   DATA[1018,16] := 1.0;
   DATA[1018,17] := 1.0;
   DATA[1018,18] := 1.0;
   DATA[1018,19] := 1.0;
   DATA[1018,20] := 148.808;
   DATA[1018,21] := 155.0115;
   DATA[1018,22] := 1.715567;
   DATA[1018,23] := 905.2679;
   DATA[1018,24] := 2.0;
   DATA[1018,25] := 2.0;
   DATA[1018,26] := 7.87798;
   DATA[1018,27] := 144.1169;
   DATA[1018,28] := 263.1056;
   DATA[1018,29] := 12.03538;
   DATA[1018,30] := 1.72443;
   DATA[1018,31] := 1.268093;
   DATA[1018,32] := 0.7351407;
   DATA[1018,33] := 0.3083624;
   DATA[1018,34] := 2.0;
   DATA[1018,35] := 250.1442;
   DATA[1018,36] := 1.649953;
   DATA[1018,37] := 189.1022;
   DATA[1018,38] := 0.000128152;
   DATA[1018,39] := 1.0;
   DATA[1019,0] := 2.541075;
   DATA[1019,1] := 664.7062;
   DATA[1019,2] := 2.0;
   DATA[1019,3] := 1.0;
   DATA[1019,4] := 262.5288;
   DATA[1019,5] := 8.462126;
   DATA[1019,6] := 315.9959;
   DATA[1019,8] := 1.0;
   DATA[1019,9] := 1.0;
   DATA[1019,10] := 1.0;
   DATA[1019,11] := 2.010372;
   DATA[1019,13] := 1011.439;
   DATA[1019,14] := 1.0;
   DATA[1019,15] := 1.0;
   DATA[1019,16] := 1.0;
   DATA[1019,17] := 1.0;
   DATA[1019,18] := 1.0;
   DATA[1019,19] := 1.0;
   DATA[1019,20] := 148.808;
   DATA[1019,21] := 155.0115;
   DATA[1019,22] := 1.715567;
   DATA[1019,23] := 904.8449;
   DATA[1019,24] := 2.0;
   DATA[1019,25] := 2.0;
   DATA[1019,26] := 7.87798;
   DATA[1019,27] := 144.0913;
   DATA[1019,28] := 263.1056;
   DATA[1019,29] := 12.03538;
   DATA[1019,30] := 1.72443;
   DATA[1019,31] := 1.265531;
   DATA[1019,32] := 0.7351407;
   DATA[1019,33] := 0.3083624;
   DATA[1019,34] := 2.0;
   DATA[1019,35] := 250.1442;
   DATA[1019,36] := 1.649953;
   DATA[1019,37] := 189.0541;
   DATA[1019,38] := 0.000128152;
   DATA[1019,39] := 1.0;
   DATA[1020,0] := 2.541075;
   DATA[1020,1] := 665.4913;
   DATA[1020,2] := 2.0;
   DATA[1020,3] := 1.0;
   DATA[1020,4] := 262.5288;
   DATA[1020,5] := 8.462126;
   DATA[1020,6] := 315.9959;
   DATA[1020,8] := 1.0;
   DATA[1020,9] := 1.0;
   DATA[1020,10] := 1.0;
   DATA[1020,11] := 2.010372;
   DATA[1020,13] := 1011.279;
   DATA[1020,14] := 1.0;
   DATA[1020,15] := 1.0;
   DATA[1020,16] := 1.0;
   DATA[1020,17] := 1.0;
   DATA[1020,18] := 1.0;
   DATA[1020,19] := 1.0;
   DATA[1020,20] := 148.808;
   DATA[1020,21] := 155.0115;
   DATA[1020,22] := 1.713645;
   DATA[1020,23] := 904.3835;
   DATA[1020,24] := 2.0;
   DATA[1020,25] := 2.0;
   DATA[1020,26] := 7.87798;
   DATA[1020,27] := 144.0913;
   DATA[1020,28] := 263.1056;
   DATA[1020,29] := 12.03538;
   DATA[1020,30] := 1.72443;
   DATA[1020,31] := 1.28436;
   DATA[1020,32] := 0.7351407;
   DATA[1020,33] := 0.3083624;
   DATA[1020,34] := 2.0;
   DATA[1020,35] := 250.1442;
   DATA[1020,36] := 1.665972;
   DATA[1020,37] := 189.0541;
   DATA[1020,38] := 0.000128152;
   DATA[1020,39] := 1.0;
   DATA[1021,0] := 2.542356;
   DATA[1021,1] := 666.4333;
   DATA[1021,2] := 2.0;
   DATA[1021,3] := 1.0;
   DATA[1021,4] := 262.5288;
   DATA[1021,5] := 8.462126;
   DATA[1021,6] := 315.8165;
   DATA[1021,8] := 1.0;
   DATA[1021,9] := 1.0;
   DATA[1021,10] := 1.0;
   DATA[1021,11] := 2.010372;
   DATA[1021,13] := 1011.279;
   DATA[1021,14] := 1.0;
   DATA[1021,15] := 1.0;
   DATA[1021,16] := 1.0;
   DATA[1021,17] := 1.0;
   DATA[1021,18] := 1.0;
   DATA[1021,19] := 1.0;
   DATA[1021,20] := 148.808;
   DATA[1021,21] := 155.0115;
   DATA[1021,22] := 1.713645;
   DATA[1021,23] := 903.8452;
   DATA[1021,24] := 2.0;
   DATA[1021,25] := 2.0;
   DATA[1021,26] := 7.87798;
   DATA[1021,27] := 144.0913;
   DATA[1021,28] := 263.1056;
   DATA[1021,29] := 12.03538;
   DATA[1021,30] := 1.72443;
   DATA[1021,31] := 1.292174;
   DATA[1021,32] := 0.7351407;
   DATA[1021,33] := 0.3083624;
   DATA[1021,34] := 2.0;
   DATA[1021,35] := 250.4005;
   DATA[1021,36] := 1.665972;
   DATA[1021,37] := 189.0541;
   DATA[1021,38] := 0.000128152;
   DATA[1021,39] := 1.0;
   DATA[1022,0] := 2.54588;
   DATA[1022,1] := 666.5511;
   DATA[1022,2] := 2.0;
   DATA[1022,3] := 1.0;
   DATA[1022,4] := 262.5288;
   DATA[1022,5] := 8.462126;
   DATA[1022,6] := 315.8165;
   DATA[1022,8] := 1.0;
   DATA[1022,9] := 1.0;
   DATA[1022,10] := 1.0;
   DATA[1022,11] := 2.010372;
   DATA[1022,13] := 1011.119;
   DATA[1022,14] := 1.0;
   DATA[1022,15] := 1.0;
   DATA[1022,16] := 1.0;
   DATA[1022,17] := 1.0;
   DATA[1022,18] := 1.0;
   DATA[1022,19] := 1.0;
   DATA[1022,20] := 148.808;
   DATA[1022,21] := 155.0115;
   DATA[1022,22] := 1.713645;
   DATA[1022,23] := 903.6913;
   DATA[1022,24] := 2.0;
   DATA[1022,25] := 2.0;
   DATA[1022,26] := 7.87798;
   DATA[1022,27] := 144.0913;
   DATA[1022,28] := 263.1056;
   DATA[1022,29] := 12.03538;
   DATA[1022,30] := 1.72443;
   DATA[1022,31] := 1.292174;
   DATA[1022,32] := 0.7351407;
   DATA[1022,33] := 0.3083624;
   DATA[1022,34] := 2.0;
   DATA[1022,35] := 250.4005;
   DATA[1022,36] := 1.69801;
   DATA[1022,37] := 189.1823;
   DATA[1022,38] := 0.000128152;
   DATA[1022,39] := 1.0;
   DATA[1023,0] := 2.54588;
   DATA[1023,1] := 667.3361;
   DATA[1023,2] := 2.0;
   DATA[1023,3] := 1.0;
   DATA[1023,4] := 262.5288;
   DATA[1023,5] := 8.462126;
   DATA[1023,6] := 315.8165;
   DATA[1023,8] := 1.0;
   DATA[1023,9] := 1.0;
   DATA[1023,10] := 1.0;
   DATA[1023,11] := 2.010372;
   DATA[1023,13] := 1011.239;
   DATA[1023,14] := 1.0;
   DATA[1023,15] := 1.0;
   DATA[1023,16] := 1.0;
   DATA[1023,17] := 1.0;
   DATA[1023,18] := 1.0;
   DATA[1023,19] := 1.0;
   DATA[1023,20] := 148.808;
   DATA[1023,21] := 155.0115;
   DATA[1023,22] := 1.716592;
   DATA[1023,23] := 903.2299;
   DATA[1023,24] := 2.0;
   DATA[1023,25] := 2.0;
   DATA[1023,26] := 7.87798;
   DATA[1023,27] := 144.0913;
   DATA[1023,28] := 263.1056;
   DATA[1023,29] := 12.03538;
   DATA[1023,30] := 1.728531;
   DATA[1023,31] := 1.292174;
   DATA[1023,32] := 0.7351407;
   DATA[1023,33] := 0.3083624;
   DATA[1023,34] := 2.0;
   DATA[1023,35] := 250.5608;
   DATA[1023,36] := 1.730048;
   DATA[1023,37] := 189.3425;
   DATA[1023,38] := 0.000128152;
   DATA[1023,39] := 1.0;
   DATA[1024,0] := 2.54588;
   DATA[1024,1] := 667.6894;
   DATA[1024,2] := 2.0;
   DATA[1024,3] := 1.0;
   DATA[1024,4] := 262.5288;
   DATA[1024,5] := 8.462126;
   DATA[1024,6] := 315.9446;
   DATA[1024,8] := 1.0;
   DATA[1024,9] := 1.0;
   DATA[1024,10] := 1.0;
   DATA[1024,11] := 2.010372;
   DATA[1024,13] := 1011.56;
   DATA[1024,14] := 1.0;
   DATA[1024,15] := 1.0;
   DATA[1024,16] := 1.0;
   DATA[1024,17] := 1.0;
   DATA[1024,18] := 1.0;
   DATA[1024,19] := 1.0;
   DATA[1024,20] := 148.808;
   DATA[1024,21] := 154.8065;
   DATA[1024,22] := 1.717746;
   DATA[1024,23] := 903.0761;
   DATA[1024,24] := 2.0;
   DATA[1024,25] := 2.0;
   DATA[1024,26] := 7.87798;
   DATA[1024,27] := 144.0913;
   DATA[1024,28] := 263.1056;
   DATA[1024,29] := 12.03538;
   DATA[1024,30] := 1.728531;
   DATA[1024,31] := 1.292174;
   DATA[1024,32] := 0.7351407;
   DATA[1024,33] := 0.3071454;
   DATA[1024,34] := 2.0;
   DATA[1024,35] := 250.5608;
   DATA[1024,36] := 1.730048;
   DATA[1024,37] := 189.3425;
   DATA[1024,38] := 0.000128152;
   DATA[1024,39] := 1.0;
   DATA[1025,0] := 2.54588;
   DATA[1025,1] := 667.6501;
   DATA[1025,2] := 2.0;
   DATA[1025,3] := 1.0;
   DATA[1025,4] := 262.5288;
   DATA[1025,5] := 8.462126;
   DATA[1025,6] := 315.9446;
   DATA[1025,8] := 1.0;
   DATA[1025,9] := 1.0;
   DATA[1025,10] := 1.0;
   DATA[1025,11] := 2.010372;
   DATA[1025,13] := 1011.56;
   DATA[1025,14] := 1.0;
   DATA[1025,15] := 1.0;
   DATA[1025,16] := 1.0;
   DATA[1025,17] := 1.0;
   DATA[1025,18] := 1.0;
   DATA[1025,19] := 1.0;
   DATA[1025,20] := 148.808;
   DATA[1025,21] := 154.8065;
   DATA[1025,22] := 1.717746;
   DATA[1025,23] := 902.4609;
   DATA[1025,24] := 2.0;
   DATA[1025,25] := 2.0;
   DATA[1025,26] := 7.87798;
   DATA[1025,27] := 144.0913;
   DATA[1025,28] := 263.1056;
   DATA[1025,29] := 12.03538;
   DATA[1025,30] := 1.726865;
   DATA[1025,31] := 1.292174;
   DATA[1025,32] := 0.7351407;
   DATA[1025,33] := 0.3068891;
   DATA[1025,34] := 2.0;
   DATA[1025,35] := 250.5608;
   DATA[1025,36] := 1.730048;
   DATA[1025,37] := 189.3425;
   DATA[1025,38] := 0.000128152;
   DATA[1025,39] := 1.0;
   DATA[1026,0] := 2.54588;
   DATA[1026,1] := 668.1997;
   DATA[1026,2] := 2.0;
   DATA[1026,3] := 1.0;
   DATA[1026,4] := 262.5288;
   DATA[1026,5] := 8.46501;
   DATA[1026,6] := 315.9446;
   DATA[1026,8] := 1.0;
   DATA[1026,9] := 1.0;
   DATA[1026,10] := 1.0;
   DATA[1026,11] := 2.010372;
   DATA[1026,13] := 1011.159;
   DATA[1026,14] := 1.0;
   DATA[1026,15] := 1.0;
   DATA[1026,16] := 1.0;
   DATA[1026,17] := 1.0;
   DATA[1026,18] := 1.0;
   DATA[1026,19] := 1.0;
   DATA[1026,20] := 148.808;
   DATA[1026,21] := 154.8065;
   DATA[1026,22] := 1.717746;
   DATA[1026,23] := 901.7688;
   DATA[1026,24] := 2.0;
   DATA[1026,25] := 2.0;
   DATA[1026,26] := 7.87798;
   DATA[1026,27] := 144.0913;
   DATA[1026,28] := 263.1056;
   DATA[1026,29] := 12.03538;
   DATA[1026,30] := 1.726224;
   DATA[1026,31] := 1.300243;
   DATA[1026,32] := 0.7351407;
   DATA[1026,33] := 0.3068891;
   DATA[1026,34] := 2.0;
   DATA[1026,35] := 250.721;
   DATA[1026,36] := 1.730048;
   DATA[1026,37] := 189.3425;
   DATA[1026,38] := 0.000128152;
   DATA[1026,39] := 1.0;
   DATA[1027,0] := 2.539474;
   DATA[1027,1] := 668.3174;
   DATA[1027,2] := 2.0;
   DATA[1027,3] := 1.0;
   DATA[1027,4] := 262.5288;
   DATA[1027,5] := 8.46501;
   DATA[1027,6] := 315.9446;
   DATA[1027,8] := 1.0;
   DATA[1027,9] := 1.0;
   DATA[1027,10] := 1.0;
   DATA[1027,11] := 2.010372;
   DATA[1027,13] := 1010.959;
   DATA[1027,14] := 1.0;
   DATA[1027,15] := 1.0;
   DATA[1027,16] := 1.0;
   DATA[1027,17] := 1.0;
   DATA[1027,18] := 1.0;
   DATA[1027,19] := 1.0;
   DATA[1027,20] := 148.808;
   DATA[1027,21] := 154.8065;
   DATA[1027,22] := 1.718643;
   DATA[1027,23] := 901.1536;
   DATA[1027,24] := 2.0;
   DATA[1027,25] := 2.0;
   DATA[1027,26] := 7.87798;
   DATA[1027,27] := 144.0913;
   DATA[1027,28] := 263.1056;
   DATA[1027,29] := 12.03538;
   DATA[1027,30] := 1.726224;
   DATA[1027,31] := 1.296657;
   DATA[1027,32] := 0.7351407;
   DATA[1027,33] := 0.3068891;
   DATA[1027,34] := 2.0;
   DATA[1027,35] := 250.753;
   DATA[1027,36] := 1.730048;
   DATA[1027,37] := 189.3425;
   DATA[1027,38] := 0.000128152;
   DATA[1027,39] := 1.0;
   DATA[1028,0] := 2.536912;
   DATA[1028,1] := 668.239;
   DATA[1028,2] := 2.0;
   DATA[1028,3] := 1.0;
   DATA[1028,4] := 262.5288;
   DATA[1028,5] := 8.46501;
   DATA[1028,6] := 315.9446;
   DATA[1028,8] := 1.0;
   DATA[1028,9] := 1.0;
   DATA[1028,10] := 1.0;
   DATA[1028,11] := 2.010372;
   DATA[1028,13] := 1011.039;
   DATA[1028,14] := 1.0;
   DATA[1028,15] := 1.0;
   DATA[1028,16] := 1.0;
   DATA[1028,17] := 1.0;
   DATA[1028,18] := 1.0;
   DATA[1028,19] := 1.0;
   DATA[1028,20] := 148.808;
   DATA[1028,21] := 154.8065;
   DATA[1028,22] := 1.720437;
   DATA[1028,23] := 901.0382;
   DATA[1028,24] := 2.0;
   DATA[1028,25] := 2.0;
   DATA[1028,26] := 7.87798;
   DATA[1028,27] := 144.0913;
   DATA[1028,28] := 263.1056;
   DATA[1028,29] := 12.03538;
   DATA[1028,30] := 1.726224;
   DATA[1028,31] := 1.291918;
   DATA[1028,32] := 0.7351407;
   DATA[1028,33] := 0.3068891;
   DATA[1028,34] := 2.0;
   DATA[1028,35] := 250.8011;
   DATA[1028,36] := 1.730048;
   DATA[1028,37] := 189.4867;
   DATA[1028,38] := 0.000128152;
   DATA[1028,39] := 1.0;
   DATA[1029,0] := 2.532428;
   DATA[1029,1] := 668.5137;
   DATA[1029,2] := 2.0;
   DATA[1029,3] := 1.0;
   DATA[1029,4] := 262.5288;
   DATA[1029,5] := 8.46501;
   DATA[1029,6] := 315.9446;
   DATA[1029,8] := 1.0;
   DATA[1029,9] := 1.0;
   DATA[1029,10] := 1.0;
   DATA[1029,11] := 2.010372;
   DATA[1029,13] := 1010.879;
   DATA[1029,14] := 1.0;
   DATA[1029,15] := 1.0;
   DATA[1029,16] := 1.0;
   DATA[1029,17] := 1.0;
   DATA[1029,18] := 1.0;
   DATA[1029,19] := 1.0;
   DATA[1029,20] := 148.808;
   DATA[1029,21] := 154.8065;
   DATA[1029,22] := 1.720565;
   DATA[1029,23] := 900.0769;
   DATA[1029,24] := 2.0;
   DATA[1029,25] := 2.0;
   DATA[1029,26] := 7.87798;
   DATA[1029,27] := 144.0913;
   DATA[1029,28] := 263.1056;
   DATA[1029,29] := 12.03538;
   DATA[1029,30] := 1.727634;
   DATA[1029,31] := 1.282311;
   DATA[1029,32] := 0.7351407;
   DATA[1029,33] := 0.3065689;
   DATA[1029,34] := 2.0;
   DATA[1029,35] := 250.8011;
   DATA[1029,36] := 1.730048;
   DATA[1029,37] := 189.5187;
   DATA[1029,38] := 0.000128152;
   DATA[1029,39] := 1.0;
   DATA[1030,0] := 2.532428;
   DATA[1030,1] := 669.2203;
   DATA[1030,2] := 2.0;
   DATA[1030,3] := 1.0;
   DATA[1030,4] := 262.5288;
   DATA[1030,5] := 8.46501;
   DATA[1030,6] := 315.9446;
   DATA[1030,8] := 1.0;
   DATA[1030,9] := 1.0;
   DATA[1030,10] := 1.0;
   DATA[1030,11] := 2.010372;
   DATA[1030,13] := 1010.879;
   DATA[1030,14] := 1.0;
   DATA[1030,15] := 1.0;
   DATA[1030,16] := 1.0;
   DATA[1030,17] := 1.0;
   DATA[1030,18] := 1.0;
   DATA[1030,19] := 1.0;
   DATA[1030,20] := 148.808;
   DATA[1030,21] := 154.6526;
   DATA[1030,22] := 1.720565;
   DATA[1030,23] := 899.5001;
   DATA[1030,24] := 2.0;
   DATA[1030,25] := 2.0;
   DATA[1030,26] := 7.87798;
   DATA[1030,27] := 144.0913;
   DATA[1030,28] := 263.1056;
   DATA[1030,29] := 12.03538;
   DATA[1030,30] := 1.727634;
   DATA[1030,31] := 1.281927;
   DATA[1030,32] := 0.7351407;
   DATA[1030,33] := 0.3065689;
   DATA[1030,34] := 2.0;
   DATA[1030,35] := 250.8011;
   DATA[1030,36] := 1.730048;
   DATA[1030,37] := 189.6148;
   DATA[1030,38] := 0.000128152;
   DATA[1030,39] := 1.0;
   DATA[1031,0] := 2.532428;
   DATA[1031,1] := 669.5735;
   DATA[1031,2] := 2.0;
   DATA[1031,3] := 1.0;
   DATA[1031,4] := 262.5288;
   DATA[1031,5] := 8.464048;
   DATA[1031,6] := 315.9446;
   DATA[1031,8] := 1.0;
   DATA[1031,9] := 1.0;
   DATA[1031,10] := 1.0;
   DATA[1031,11] := 2.010372;
   DATA[1031,13] := 1010.959;
   DATA[1031,14] := 1.0;
   DATA[1031,15] := 1.0;
   DATA[1031,16] := 1.0;
   DATA[1031,17] := 1.0;
   DATA[1031,18] := 1.0;
   DATA[1031,19] := 1.0;
   DATA[1031,20] := 148.808;
   DATA[1031,21] := 154.6526;
   DATA[1031,22] := 1.720565;
   DATA[1031,23] := 899.2694;
   DATA[1031,24] := 2.0;
   DATA[1031,25] := 2.0;
   DATA[1031,26] := 7.87798;
   DATA[1031,27] := 144.0913;
   DATA[1031,28] := 263.1056;
   DATA[1031,29] := 12.03538;
   DATA[1031,30] := 1.727634;
   DATA[1031,31] := 1.286922;
   DATA[1031,32] := 0.7351407;
   DATA[1031,33] := 0.3065689;
   DATA[1031,34] := 2.0;
   DATA[1031,35] := 250.8011;
   DATA[1031,36] := 1.730048;
   DATA[1031,37] := 189.6148;
   DATA[1031,38] := 0.000128152;
   DATA[1031,39] := 1.0;
   DATA[1032,0] := 2.538513;
   DATA[1032,1] := 669.652;
   DATA[1032,2] := 2.0;
   DATA[1032,3] := 1.0;
   DATA[1032,4] := 262.5288;
   DATA[1032,5] := 8.462446;
   DATA[1032,6] := 316.0728;
   DATA[1032,8] := 1.0;
   DATA[1032,9] := 1.0;
   DATA[1032,10] := 1.0;
   DATA[1032,11] := 2.010372;
   DATA[1032,13] := 1011.079;
   DATA[1032,14] := 1.0;
   DATA[1032,15] := 1.0;
   DATA[1032,16] := 1.0;
   DATA[1032,17] := 1.0;
   DATA[1032,18] := 1.0;
   DATA[1032,19] := 1.0;
   DATA[1032,20] := 148.808;
   DATA[1032,21] := 154.6526;
   DATA[1032,22] := 1.719668;
   DATA[1032,23] := 899.0002;
   DATA[1032,24] := 2.0;
   DATA[1032,25] := 2.0;
   DATA[1032,26] := 7.87798;
   DATA[1032,27] := 144.0913;
   DATA[1032,28] := 263.1056;
   DATA[1032,29] := 12.03538;
   DATA[1032,30] := 1.727634;
   DATA[1032,31] := 1.29243;
   DATA[1032,32] := 0.7351407;
   DATA[1032,33] := 0.3065689;
   DATA[1032,34] := 2.0;
   DATA[1032,35] := 250.8652;
   DATA[1032,36] := 1.730048;
   DATA[1032,37] := 189.6148;
   DATA[1032,38] := 0.000128152;
   DATA[1032,39] := 1.0;
   DATA[1033,0] := 2.543638;
   DATA[1033,1] := 670.0839;
   DATA[1033,2] := 2.0;
   DATA[1033,3] := 1.0;
   DATA[1033,4] := 262.5288;
   DATA[1033,5] := 8.461164;
   DATA[1033,6] := 316.0728;
   DATA[1033,8] := 1.0;
   DATA[1033,9] := 1.0;
   DATA[1033,10] := 1.0;
   DATA[1033,11] := 2.010372;
   DATA[1033,13] := 1010.959;
   DATA[1033,14] := 1.0;
   DATA[1033,15] := 1.0;
   DATA[1033,16] := 1.0;
   DATA[1033,17] := 1.0;
   DATA[1033,18] := 1.0;
   DATA[1033,19] := 1.0;
   DATA[1033,20] := 148.808;
   DATA[1033,21] := 154.6526;
   DATA[1033,22] := 1.718643;
   DATA[1033,23] := 898.4619;
   DATA[1033,24] := 2.0;
   DATA[1033,25] := 2.0;
   DATA[1033,26] := 7.87798;
   DATA[1033,27] := 144.0913;
   DATA[1033,28] := 263.1056;
   DATA[1033,29] := 12.03538;
   DATA[1033,30] := 1.72789;
   DATA[1033,31] := 1.29243;
   DATA[1033,32] := 0.7351407;
   DATA[1033,33] := 0.3065689;
   DATA[1033,34] := 2.0;
   DATA[1033,35] := 250.9453;
   DATA[1033,36] := 1.730048;
   DATA[1033,37] := 189.6148;
   DATA[1033,38] := 0.000128152;
   DATA[1033,39] := 1.0;
   DATA[1034,0] := 2.54684;
   DATA[1034,1] := 671.1437;
   DATA[1034,2] := 2.0;
   DATA[1034,3] := 1.0;
   DATA[1034,4] := 262.5288;
   DATA[1034,5] := 8.461164;
   DATA[1034,6] := 316.0728;
   DATA[1034,8] := 1.0;
   DATA[1034,9] := 1.0;
   DATA[1034,10] := 1.0;
   DATA[1034,11] := 2.010372;
   DATA[1034,13] := 1011.039;
   DATA[1034,14] := 1.0;
   DATA[1034,15] := 1.0;
   DATA[1034,16] := 1.0;
   DATA[1034,17] := 1.0;
   DATA[1034,18] := 1.0;
   DATA[1034,19] := 1.0;
   DATA[1034,20] := 148.808;
   DATA[1034,21] := 154.8321;
   DATA[1034,22] := 1.718643;
   DATA[1034,23] := 898.0389;
   DATA[1034,24] := 2.0;
   DATA[1034,25] := 2.0;
   DATA[1034,26] := 7.87798;
   DATA[1034,27] := 144.0913;
   DATA[1034,28] := 263.1056;
   DATA[1034,29] := 12.03538;
   DATA[1034,30] := 1.728788;
   DATA[1034,31] := 1.283592;
   DATA[1034,32] := 0.7351407;
   DATA[1034,33] := 0.3065689;
   DATA[1034,34] := 2.0;
   DATA[1034,35] := 250.9453;
   DATA[1034,36] := 1.730048;
   DATA[1034,37] := 189.6148;
   DATA[1034,38] := 0.000128152;
   DATA[1034,39] := 1.0;
   DATA[1035,0] := 2.54684;
   DATA[1035,1] := 671.811;
   DATA[1035,2] := 2.0;
   DATA[1035,3] := 1.0;
   DATA[1035,4] := 262.5288;
   DATA[1035,5] := 8.461164;
   DATA[1035,6] := 316.0728;
   DATA[1035,8] := 1.0;
   DATA[1035,9] := 1.0;
   DATA[1035,10] := 1.0;
   DATA[1035,11] := 2.010372;
   DATA[1035,13] := 1010.919;
   DATA[1035,14] := 1.0;
   DATA[1035,15] := 1.0;
   DATA[1035,16] := 1.0;
   DATA[1035,17] := 1.0;
   DATA[1035,18] := 1.0;
   DATA[1035,19] := 1.0;
   DATA[1035,20] := 148.808;
   DATA[1035,21] := 154.8321;
   DATA[1035,22] := 1.719796;
   DATA[1035,23] := 897.8467;
   DATA[1035,24] := 2.0;
   DATA[1035,25] := 2.0;
   DATA[1035,26] := 7.87798;
   DATA[1035,27] := 144.0913;
   DATA[1035,28] := 263.1056;
   DATA[1035,29] := 12.03538;
   DATA[1035,30] := 1.729428;
   DATA[1035,31] := 1.264506;
   DATA[1035,32] := 0.7351407;
   DATA[1035,33] := 0.3065689;
   DATA[1035,34] := 2.0;
   DATA[1035,35] := 250.9453;
   DATA[1035,36] := 1.730048;
   DATA[1035,37] := 189.6148;
   DATA[1035,38] := 0.000128152;
   DATA[1035,39] := 1.0;
   DATA[1036,0] := 2.550684;
   DATA[1036,1] := 672.125;
   DATA[1036,2] := 2.0;
   DATA[1036,3] := 1.0;
   DATA[1036,4] := 262.5288;
   DATA[1036,5] := 8.461164;
   DATA[1036,6] := 316.0728;
   DATA[1036,8] := 1.0;
   DATA[1036,9] := 1.0;
   DATA[1036,10] := 1.0;
   DATA[1036,11] := 2.010372;
   DATA[1036,13] := 1010.718;
   DATA[1036,14] := 1.0;
   DATA[1036,15] := 1.0;
   DATA[1036,16] := 1.0;
   DATA[1036,17] := 1.0;
   DATA[1036,18] := 1.0;
   DATA[1036,19] := 1.0;
   DATA[1036,20] := 148.808;
   DATA[1036,21] := 154.8321;
   DATA[1036,22] := 1.719796;
   DATA[1036,23] := 897.616;
   DATA[1036,24] := 2.0;
   DATA[1036,25] := 2.0;
   DATA[1036,26] := 7.87798;
   DATA[1036,27] := 144.0913;
   DATA[1036,28] := 263.1056;
   DATA[1036,29] := 12.03538;
   DATA[1036,30] := 1.729428;
   DATA[1036,31] := 1.262457;
   DATA[1036,32] := 0.7351407;
   DATA[1036,33] := 0.3065689;
   DATA[1036,34] := 2.0;
   DATA[1036,35] := 250.9453;
   DATA[1036,36] := 1.730048;
   DATA[1036,37] := 189.6148;
   DATA[1036,38] := 0.000128152;
   DATA[1036,39] := 1.0;
   DATA[1037,0] := 2.550684;
   DATA[1037,1] := 673.0278;
   DATA[1037,2] := 2.0;
   DATA[1037,3] := 1.0;
   DATA[1037,4] := 262.5288;
   DATA[1037,5] := 8.461164;
   DATA[1037,6] := 316.201;
   DATA[1037,8] := 1.0;
   DATA[1037,9] := 1.0;
   DATA[1037,10] := 1.0;
   DATA[1037,11] := 2.010372;
   DATA[1037,13] := 1011.279;
   DATA[1037,14] := 1.0;
   DATA[1037,15] := 1.0;
   DATA[1037,16] := 1.0;
   DATA[1037,17] := 1.0;
   DATA[1037,18] := 1.0;
   DATA[1037,19] := 1.0;
   DATA[1037,20] := 148.808;
   DATA[1037,21] := 154.8321;
   DATA[1037,22] := 1.719796;
   DATA[1037,23] := 897.27;
   DATA[1037,24] := 2.0;
   DATA[1037,25] := 2.0;
   DATA[1037,26] := 7.87798;
   DATA[1037,27] := 144.0913;
   DATA[1037,28] := 263.1056;
   DATA[1037,29] := 12.03538;
   DATA[1037,30] := 1.729428;
   DATA[1037,31] := 1.265147;
   DATA[1037,32] := 0.7351407;
   DATA[1037,33] := 0.3080421;
   DATA[1037,34] := 2.0;
   DATA[1037,35] := 250.753;
   DATA[1037,36] := 1.730048;
   DATA[1037,37] := 189.6148;
   DATA[1037,38] := 0.000128152;
   DATA[1037,39] := 1.0;
   DATA[1038,0] := 2.550684;
   DATA[1038,1] := 673.7343;
   DATA[1038,2] := 2.0;
   DATA[1038,3] := 1.0;
   DATA[1038,4] := 262.5288;
   DATA[1038,5] := 8.463408;
   DATA[1038,6] := 316.201;
   DATA[1038,8] := 1.0;
   DATA[1038,9] := 1.0;
   DATA[1038,10] := 1.0;
   DATA[1038,11] := 2.010372;
   DATA[1038,13] := 1011.159;
   DATA[1038,14] := 1.0;
   DATA[1038,15] := 1.0;
   DATA[1038,16] := 1.0;
   DATA[1038,17] := 1.0;
   DATA[1038,18] := 1.0;
   DATA[1038,19] := 1.0;
   DATA[1038,20] := 148.808;
   DATA[1038,21] := 154.8321;
   DATA[1038,22] := 1.717361;
   DATA[1038,23] := 897.2315;
   DATA[1038,24] := 2.0;
   DATA[1038,25] := 2.0;
   DATA[1038,26] := 7.87798;
   DATA[1038,27] := 144.0913;
   DATA[1038,28] := 263.1056;
   DATA[1038,29] := 12.03538;
   DATA[1038,30] := 1.729428;
   DATA[1038,31] := 1.272704;
   DATA[1038,32] := 0.7351407;
   DATA[1038,33] := 0.3082983;
   DATA[1038,34] := 2.0;
   DATA[1038,35] := 250.6569;
   DATA[1038,36] := 1.730048;
   DATA[1038,37] := 189.6148;
   DATA[1038,38] := 0.000128152;
   DATA[1038,39] := 1.0;
   DATA[1039,0] := 2.543958;
   DATA[1039,1] := 673.8914;
   DATA[1039,2] := 2.0;
   DATA[1039,3] := 1.0;
   DATA[1039,4] := 262.5288;
   DATA[1039,5] := 8.464369;
   DATA[1039,6] := 316.201;
   DATA[1039,8] := 1.0;
   DATA[1039,9] := 1.0;
   DATA[1039,10] := 1.0;
   DATA[1039,11] := 2.010372;
   DATA[1039,13] := 1011.479;
   DATA[1039,14] := 1.0;
   DATA[1039,15] := 1.0;
   DATA[1039,16] := 1.0;
   DATA[1039,17] := 1.0;
   DATA[1039,18] := 1.0;
   DATA[1039,19] := 1.0;
   DATA[1039,20] := 148.808;
   DATA[1039,21] := 154.8321;
   DATA[1039,22] := 1.717361;
   DATA[1039,23] := 896.9623;
   DATA[1039,24] := 2.0;
   DATA[1039,25] := 2.0;
   DATA[1039,26] := 7.87798;
   DATA[1039,27] := 144.0913;
   DATA[1039,28] := 263.1056;
   DATA[1039,29] := 12.03538;
   DATA[1039,30] := 1.7293;
   DATA[1039,31] := 1.281927;
   DATA[1039,32] := 0.7352687;
   DATA[1039,33] := 0.3082983;
   DATA[1039,34] := 2.0;
   DATA[1039,35] := 250.6569;
   DATA[1039,36] := 1.681991;
   DATA[1039,37] := 189.6148;
   DATA[1039,38] := 0.000128152;
   DATA[1039,39] := 1.0;
   DATA[1040,0] := 2.543958;
   DATA[1040,1] := 674.5194;
   DATA[1040,2] := 2.0;
   DATA[1040,3] := 1.0;
   DATA[1040,4] := 262.5288;
   DATA[1040,5] := 8.464369;
   DATA[1040,6] := 316.201;
   DATA[1040,8] := 1.0;
   DATA[1040,9] := 1.0;
   DATA[1040,10] := 1.0;
   DATA[1040,11] := 2.010372;
   DATA[1040,13] := 1011.119;
   DATA[1040,14] := 1.0;
   DATA[1040,15] := 1.0;
   DATA[1040,16] := 1.0;
   DATA[1040,17] := 1.0;
   DATA[1040,18] := 1.0;
   DATA[1040,19] := 1.0;
   DATA[1040,20] := 148.808;
   DATA[1040,21] := 154.8321;
   DATA[1040,22] := 1.717361;
   DATA[1040,23] := 896.6932;
   DATA[1040,24] := 2.0;
   DATA[1040,25] := 2.0;
   DATA[1040,26] := 7.87798;
   DATA[1040,27] := 144.0913;
   DATA[1040,28] := 263.1056;
   DATA[1040,29] := 12.03538;
   DATA[1040,30] := 1.728659;
   DATA[1040,31] := 1.282439;
   DATA[1040,32] := 0.7353967;
   DATA[1040,33] := 0.3082983;
   DATA[1040,34] := 2.0;
   DATA[1040,35] := 250.6569;
   DATA[1040,36] := 1.681991;
   DATA[1040,37] := 189.3745;
   DATA[1040,38] := 0.000128152;
   DATA[1040,39] := 1.0;
   DATA[1041,0] := 2.542356;
   DATA[1041,1] := 675.1082;
   DATA[1041,2] := 2.0;
   DATA[1041,3] := 1.0;
   DATA[1041,4] := 262.5288;
   DATA[1041,5] := 8.464369;
   DATA[1041,6] := 316.201;
   DATA[1041,8] := 1.0;
   DATA[1041,9] := 1.0;
   DATA[1041,10] := 1.0;
   DATA[1041,11] := 2.010372;
   DATA[1041,13] := 1011.319;
   DATA[1041,14] := 1.0;
   DATA[1041,15] := 1.0;
   DATA[1041,16] := 1.0;
   DATA[1041,17] := 1.0;
   DATA[1041,18] := 1.0;
   DATA[1041,19] := 1.0;
   DATA[1041,20] := 148.808;
   DATA[1041,21] := 154.8321;
   DATA[1041,22] := 1.717361;
   DATA[1041,23] := 896.3856;
   DATA[1041,24] := 2.0;
   DATA[1041,25] := 2.0;
   DATA[1041,26] := 7.87798;
   DATA[1041,27] := 144.0913;
   DATA[1041,28] := 263.1056;
   DATA[1041,29] := 12.03538;
   DATA[1041,30] := 1.726737;
   DATA[1041,31] := 1.274625;
   DATA[1041,32] := 0.7353967;
   DATA[1041,33] := 0.3082983;
   DATA[1041,34] := 2.0;
   DATA[1041,35] := 250.6569;
   DATA[1041,36] := 1.681991;
   DATA[1041,37] := 189.3745;
   DATA[1041,38] := 0.000128152;
   DATA[1041,39] := 1.0;
   DATA[1042,0] := 2.541075;
   DATA[1042,1] := 676.0502;
   DATA[1042,2] := 2.0;
   DATA[1042,3] := 1.0;
   DATA[1042,4] := 262.5288;
   DATA[1042,5] := 8.464369;
   DATA[1042,6] := 316.201;
   DATA[1042,8] := 1.0;
   DATA[1042,9] := 1.0;
   DATA[1042,10] := 1.0;
   DATA[1042,11] := 2.010372;
   DATA[1042,13] := 1011.039;
   DATA[1042,14] := 1.0;
   DATA[1042,15] := 1.0;
   DATA[1042,16] := 1.0;
   DATA[1042,17] := 1.0;
   DATA[1042,18] := 1.0;
   DATA[1042,19] := 1.0;
   DATA[1042,20] := 148.808;
   DATA[1042,21] := 154.8321;
   DATA[1042,22] := 1.718387;
   DATA[1042,23] := 895.8088;
   DATA[1042,24] := 2.0;
   DATA[1042,25] := 2.0;
   DATA[1042,26] := 7.87798;
   DATA[1042,27] := 144.0913;
   DATA[1042,28] := 263.1056;
   DATA[1042,29] := 12.03538;
   DATA[1042,30] := 1.72443;
   DATA[1042,31] := 1.279237;
   DATA[1042,32] := 0.7353967;
   DATA[1042,33] := 0.3082983;
   DATA[1042,34] := 2.0;
   DATA[1042,35] := 250.6569;
   DATA[1042,36] := 1.681991;
   DATA[1042,37] := 189.3745;
   DATA[1042,38] := 0.000128152;
   DATA[1042,39] := 1.0;
   DATA[1043,0] := 2.540435;
   DATA[1043,1] := 676.5605;
   DATA[1043,2] := 2.0;
   DATA[1043,3] := 1.0;
   DATA[1043,4] := 262.5288;
   DATA[1043,5] := 8.464369;
   DATA[1043,6] := 316.201;
   DATA[1043,8] := 1.0;
   DATA[1043,9] := 1.0;
   DATA[1043,10] := 1.0;
   DATA[1043,11] := 2.010372;
   DATA[1043,13] := 1010.638;
   DATA[1043,14] := 1.0;
   DATA[1043,15] := 1.0;
   DATA[1043,16] := 1.0;
   DATA[1043,17] := 1.0;
   DATA[1043,18] := 1.0;
   DATA[1043,19] := 1.0;
   DATA[1043,20] := 148.808;
   DATA[1043,21] := 154.8321;
   DATA[1043,22] := 1.718515;
   DATA[1043,23] := 895.6165;
   DATA[1043,24] := 2.0;
   DATA[1043,25] := 2.0;
   DATA[1043,26] := 7.87798;
   DATA[1043,27] := 144.0656;
   DATA[1043,28] := 263.1056;
   DATA[1043,29] := 12.03538;
   DATA[1043,30] := 1.72443;
   DATA[1043,31] := 1.280902;
   DATA[1043,32] := 0.7353967;
   DATA[1043,33] := 0.3082983;
   DATA[1043,34] := 2.0;
   DATA[1043,35] := 250.6569;
   DATA[1043,36] := 1.681991;
   DATA[1043,37] := 189.3745;
   DATA[1043,38] := 0.000128152;
   DATA[1043,39] := 1.0;
   DATA[1044,0] := 2.540435;
   DATA[1044,1] := 677.2671;
   DATA[1044,2] := 2.0;
   DATA[1044,3] := 1.0;
   DATA[1044,4] := 262.5288;
   DATA[1044,5] := 8.464369;
   DATA[1044,6] := 316.201;
   DATA[1044,8] := 1.0;
   DATA[1044,9] := 1.0;
   DATA[1044,10] := 1.0;
   DATA[1044,11] := 2.010372;
   DATA[1044,13] := 1010.879;
   DATA[1044,14] := 1.0;
   DATA[1044,15] := 1.0;
   DATA[1044,16] := 1.0;
   DATA[1044,17] := 1.0;
   DATA[1044,18] := 1.0;
   DATA[1044,19] := 1.0;
   DATA[1044,20] := 148.808;
   DATA[1044,21] := 154.8321;
   DATA[1044,22] := 1.718515;
   DATA[1044,23] := 895.3858;
   DATA[1044,24] := 2.0;
   DATA[1044,25] := 2.0;
   DATA[1044,26] := 7.87798;
   DATA[1044,27] := 143.8093;
   DATA[1044,28] := 263.1056;
   DATA[1044,29] := 12.03538;
   DATA[1044,30] := 1.726096;
   DATA[1044,31] := 1.272576;
   DATA[1044,32] := 0.7353967;
   DATA[1044,33] := 0.3082983;
   DATA[1044,34] := 2.0;
   DATA[1044,35] := 250.5768;
   DATA[1044,36] := 1.681991;
   DATA[1044,37] := 189.3745;
   DATA[1044,38] := 0.000128152;
   DATA[1044,39] := 1.0;
   DATA[1045,0] := 2.54588;
   DATA[1045,1] := 678.2877;
   DATA[1045,2] := 2.0;
   DATA[1045,3] := 1.0;
   DATA[1045,4] := 262.5288;
   DATA[1045,5] := 8.464369;
   DATA[1045,6] := 316.201;
   DATA[1045,8] := 1.0;
   DATA[1045,9] := 1.0;
   DATA[1045,10] := 1.0;
   DATA[1045,11] := 2.010372;
   DATA[1045,13] := 1010.758;
   DATA[1045,14] := 1.0;
   DATA[1045,15] := 1.0;
   DATA[1045,16] := 1.0;
   DATA[1045,17] := 1.0;
   DATA[1045,18] := 1.0;
   DATA[1045,19] := 1.0;
   DATA[1045,20] := 148.808;
   DATA[1045,21] := 154.8321;
   DATA[1045,22] := 1.718515;
   DATA[1045,23] := 894.7706;
   DATA[1045,24] := 2.0;
   DATA[1045,25] := 2.0;
   DATA[1045,26] := 7.87798;
   DATA[1045,27] := 143.8093;
   DATA[1045,28] := 263.1056;
   DATA[1045,29] := 12.03538;
   DATA[1045,30] := 1.727378;
   DATA[1045,31] := 1.262329;
   DATA[1045,32] := 0.7353967;
   DATA[1045,33] := 0.3082983;
   DATA[1045,34] := 2.0;
   DATA[1045,35] := 250.5127;
   DATA[1045,36] := 1.681991;
   DATA[1045,37] := 189.3745;
   DATA[1045,38] := 0.000128152;
   DATA[1045,39] := 1.0;
   DATA[1046,0] := 2.54588;
   DATA[1046,1] := 678.9942;
   DATA[1046,2] := 2.0;
   DATA[1046,3] := 1.0;
   DATA[1046,4] := 262.5288;
   DATA[1046,5] := 8.464369;
   DATA[1046,6] := 316.201;
   DATA[1046,8] := 1.0;
   DATA[1046,9] := 1.0;
   DATA[1046,10] := 1.0;
   DATA[1046,11] := 2.010372;
   DATA[1046,13] := 1010.839;
   DATA[1046,14] := 1.0;
   DATA[1046,15] := 1.0;
   DATA[1046,16] := 1.0;
   DATA[1046,17] := 1.0;
   DATA[1046,18] := 1.0;
   DATA[1046,19] := 1.0;
   DATA[1046,20] := 148.808;
   DATA[1046,21] := 154.8321;
   DATA[1046,22] := 1.717746;
   DATA[1046,23] := 894.386;
   DATA[1046,24] := 2.0;
   DATA[1046,25] := 2.0;
   DATA[1046,26] := 7.87798;
   DATA[1046,27] := 143.8093;
   DATA[1046,28] := 263.1056;
   DATA[1046,29] := 12.03538;
   DATA[1046,30] := 1.727378;
   DATA[1046,31] := 1.261176;
   DATA[1046,32] := 0.7353967;
   DATA[1046,33] := 0.3082983;
   DATA[1046,34] := 2.0;
   DATA[1046,35] := 250.4967;
   DATA[1046,36] := 1.681991;
   DATA[1046,37] := 189.3745;
   DATA[1046,38] := 0.000128152;
   DATA[1046,39] := 1.0;
   DATA[1047,0] := 2.550364;
   DATA[1047,1] := 679.2297;
   DATA[1047,2] := 2.0;
   DATA[1047,3] := 1.0;
   DATA[1047,4] := 262.5288;
   DATA[1047,5] := 8.464369;
   DATA[1047,6] := 316.201;
   DATA[1047,8] := 1.0;
   DATA[1047,9] := 1.0;
   DATA[1047,10] := 1.0;
   DATA[1047,11] := 2.010372;
   DATA[1047,13] := 1010.558;
   DATA[1047,14] := 1.0;
   DATA[1047,15] := 1.0;
   DATA[1047,16] := 1.0;
   DATA[1047,17] := 1.0;
   DATA[1047,18] := 1.0;
   DATA[1047,19] := 1.0;
   DATA[1047,20] := 148.808;
   DATA[1047,21] := 154.8321;
   DATA[1047,22] := 1.717746;
   DATA[1047,23] := 894.1938;
   DATA[1047,24] := 2.0;
   DATA[1047,25] := 2.0;
   DATA[1047,26] := 7.87798;
   DATA[1047,27] := 143.8093;
   DATA[1047,28] := 263.1056;
   DATA[1047,29] := 12.03538;
   DATA[1047,30] := 1.727378;
   DATA[1047,31] := 1.265147;
   DATA[1047,32] := 0.7353967;
   DATA[1047,33] := 0.3082983;
   DATA[1047,34] := 2.0;
   DATA[1047,35] := 250.4326;
   DATA[1047,36] := 1.601897;
   DATA[1047,37] := 189.3745;
   DATA[1047,38] := 0.000128152;
   DATA[1047,39] := 1.0;
   DATA[1048,0] := 2.551965;
   DATA[1048,1] := 679.583;
   DATA[1048,2] := 2.0;
   DATA[1048,3] := 1.0;
   DATA[1048,4] := 262.5288;
   DATA[1048,5] := 8.462767;
   DATA[1048,6] := 316.201;
   DATA[1048,8] := 1.0;
   DATA[1048,9] := 1.0;
   DATA[1048,10] := 1.0;
   DATA[1048,11] := 2.000768;
   DATA[1048,13] := 1010.919;
   DATA[1048,14] := 1.0;
   DATA[1048,15] := 1.0;
   DATA[1048,16] := 1.0;
   DATA[1048,17] := 1.0;
   DATA[1048,18] := 1.0;
   DATA[1048,19] := 1.0;
   DATA[1048,20] := 148.808;
   DATA[1048,21] := 154.8321;
   DATA[1048,22] := 1.717746;
   DATA[1048,23] := 894.0015;
   DATA[1048,24] := 2.0;
   DATA[1048,25] := 2.0;
   DATA[1048,26] := 7.87798;
   DATA[1048,27] := 143.8093;
   DATA[1048,28] := 263.1056;
   DATA[1048,29] := 12.03538;
   DATA[1048,30] := 1.724686;
   DATA[1048,31] := 1.291533;
   DATA[1048,32] := 0.7353967;
   DATA[1048,33] := 0.3082983;
   DATA[1048,34] := 2.0;
   DATA[1048,35] := 250.4326;
   DATA[1048,36] := 1.601897;
   DATA[1048,37] := 189.2944;
   DATA[1048,38] := 0.000128152;
   DATA[1048,39] := 1.0;
   DATA[1049,0] := 2.551965;
   DATA[1049,1] := 679.6615;
   DATA[1049,2] := 2.0;
   DATA[1049,3] := 1.0;
   DATA[1049,4] := 262.5288;
   DATA[1049,5] := 8.462767;
   DATA[1049,6] := 316.201;
   DATA[1049,8] := 1.0;
   DATA[1049,9] := 1.0;
   DATA[1049,10] := 1.0;
   DATA[1049,11] := 2.000768;
   DATA[1049,13] := 1010.678;
   DATA[1049,14] := 1.0;
   DATA[1049,15] := 1.0;
   DATA[1049,16] := 1.0;
   DATA[1049,17] := 1.0;
   DATA[1049,18] := 1.0;
   DATA[1049,19] := 1.0;
   DATA[1049,20] := 148.808;
   DATA[1049,21] := 154.8321;
   DATA[1049,22] := 1.717746;
   DATA[1049,23] := 893.6939;
   DATA[1049,24] := 2.0;
   DATA[1049,25] := 2.0;
   DATA[1049,26] := 7.87798;
   DATA[1049,27] := 143.8093;
   DATA[1049,28] := 263.1056;
   DATA[1049,29] := 12.03538;
   DATA[1049,30] := 1.724301;
   DATA[1049,31] := 1.306008;
   DATA[1049,32] := 0.7353967;
   DATA[1049,33] := 0.3082983;
   DATA[1049,34] := 2.0;
   DATA[1049,35] := 250.4326;
   DATA[1049,36] := 1.601897;
   DATA[1049,37] := 189.2624;
   DATA[1049,38] := 0.000128152;
   DATA[1049,39] := 1.0;
   DATA[1050,0] := 2.548121;
   DATA[1050,1] := 679.9755;
   DATA[1050,2] := 2.0;
   DATA[1050,3] := 1.0;
   DATA[1050,4] := 262.5288;
   DATA[1050,5] := 8.461164;
   DATA[1050,6] := 316.201;
   DATA[1050,8] := 1.0;
   DATA[1050,9] := 1.0;
   DATA[1050,10] := 1.0;
   DATA[1050,11] := 2.000768;
   DATA[1050,13] := 1010.959;
   DATA[1050,14] := 1.0;
   DATA[1050,15] := 1.0;
   DATA[1050,16] := 1.0;
   DATA[1050,17] := 1.0;
   DATA[1050,18] := 1.0;
   DATA[1050,19] := 1.0;
   DATA[1050,20] := 148.808;
   DATA[1050,21] := 154.8321;
   DATA[1050,22] := 1.715824;
   DATA[1050,23] := 893.3094;
   DATA[1050,24] := 2.0;
   DATA[1050,25] := 2.0;
   DATA[1050,26] := 7.87798;
   DATA[1050,27] := 143.8093;
   DATA[1050,28] := 263.1056;
   DATA[1050,29] := 12.03538;
   DATA[1050,30] := 1.724301;
   DATA[1050,31] := 1.302293;
   DATA[1050,32] := 0.7353967;
   DATA[1050,33] := 0.3082983;
   DATA[1050,34] := 2.0;
   DATA[1050,35] := 250.2724;
   DATA[1050,36] := 1.601897;
   DATA[1050,37] := 189.1182;
   DATA[1050,38] := 0.000128152;
   DATA[1050,39] := 1.0;
   DATA[1051,0] := 2.543317;
   DATA[1051,1] := 680.5643;
   DATA[1051,2] := 2.0;
   DATA[1051,3] := 1.0;
   DATA[1051,4] := 262.5288;
   DATA[1051,5] := 8.461164;
   DATA[1051,6] := 316.201;
   DATA[1051,8] := 1.0;
   DATA[1051,9] := 1.0;
   DATA[1051,10] := 1.0;
   DATA[1051,11] := 2.000768;
   DATA[1051,13] := 1011.319;
   DATA[1051,14] := 1.0;
   DATA[1051,15] := 1.0;
   DATA[1051,16] := 1.0;
   DATA[1051,17] := 1.0;
   DATA[1051,18] := 1.0;
   DATA[1051,19] := 1.0;
   DATA[1051,20] := 148.808;
   DATA[1051,21] := 154.8321;
   DATA[1051,22] := 1.715824;
   DATA[1051,23] := 892.8864;
   DATA[1051,24] := 2.0;
   DATA[1051,25] := 2.0;
   DATA[1051,26] := 7.87798;
   DATA[1051,27] := 143.8093;
   DATA[1051,28] := 263.1056;
   DATA[1051,29] := 12.03538;
   DATA[1051,30] := 1.725327;
   DATA[1051,31] := 1.286666;
   DATA[1051,32] := 0.7353967;
   DATA[1051,33] := 0.3082983;
   DATA[1051,34] := 2.0;
   DATA[1051,35] := 250.2724;
   DATA[1051,36] := 1.601897;
   DATA[1051,37] := 189.1182;
   DATA[1051,38] := 0.000128152;
   DATA[1051,39] := 1.0;
   DATA[1052,0] := 2.543317;
   DATA[1052,1] := 681.3886;
   DATA[1052,2] := 2.0;
   DATA[1052,3] := 1.0;
   DATA[1052,4] := 262.5288;
   DATA[1052,5] := 8.461164;
   DATA[1052,6] := 316.201;
   DATA[1052,8] := 1.0;
   DATA[1052,9] := 1.0;
   DATA[1052,10] := 1.0;
   DATA[1052,11] := 2.000768;
   DATA[1052,13] := 1011.159;
   DATA[1052,14] := 1.0;
   DATA[1052,15] := 1.0;
   DATA[1052,16] := 1.0;
   DATA[1052,17] := 1.0;
   DATA[1052,18] := 1.0;
   DATA[1052,19] := 1.0;
   DATA[1052,20] := 148.808;
   DATA[1052,21] := 154.8321;
   DATA[1052,22] := 1.715824;
   DATA[1052,23] := 892.6172;
   DATA[1052,24] := 2.0;
   DATA[1052,25] := 2.0;
   DATA[1052,26] := 7.87798;
   DATA[1052,27] := 143.8862;
   DATA[1052,28] := 263.1056;
   DATA[1052,29] := 12.03538;
   DATA[1052,30] := 1.725327;
   DATA[1052,31] := 1.281158;
   DATA[1052,32] := 0.7353967;
   DATA[1052,33] := 0.3068891;
   DATA[1052,34] := 2.0;
   DATA[1052,35] := 250.1602;
   DATA[1052,36] := 1.665972;
   DATA[1052,37] := 189.1182;
   DATA[1052,38] := 0.000128152;
   DATA[1052,39] := 1.0;
   DATA[1053,0] := 2.540115;
   DATA[1053,1] := 681.8204;
   DATA[1053,2] := 2.0;
   DATA[1053,3] := 1.0;
   DATA[1053,4] := 262.5288;
   DATA[1053,5] := 8.461164;
   DATA[1053,6] := 316.201;
   DATA[1053,8] := 1.0;
   DATA[1053,9] := 1.0;
   DATA[1053,10] := 1.0;
   DATA[1053,11] := 2.000768;
   DATA[1053,13] := 1011.159;
   DATA[1053,14] := 1.0;
   DATA[1053,15] := 1.0;
   DATA[1053,16] := 1.0;
   DATA[1053,17] := 1.0;
   DATA[1053,18] := 1.0;
   DATA[1053,19] := 1.0;
   DATA[1053,20] := 148.808;
   DATA[1053,21] := 154.8321;
   DATA[1053,22] := 1.714158;
   DATA[1053,23] := 892.2328;
   DATA[1053,24] := 2.0;
   DATA[1053,25] := 2.0;
   DATA[1053,26] := 7.87798;
   DATA[1053,27] := 143.9375;
   DATA[1053,28] := 263.1056;
   DATA[1053,29] := 12.03538;
   DATA[1053,30] := 1.72507;
   DATA[1053,31] := 1.281158;
   DATA[1053,32] := 0.7353967;
   DATA[1053,33] := 0.3074016;
   DATA[1053,34] := 2.0;
   DATA[1053,35] := 250.1602;
   DATA[1053,36] := 1.665972;
   DATA[1053,37] := 189.0381;
   DATA[1053,38] := 0.000128152;
   DATA[1053,39] := 1.0;
   DATA[1054,0] := 2.540115;
   DATA[1054,1] := 681.8989;
   DATA[1054,2] := 2.0;
   DATA[1054,3] := 1.0;
   DATA[1054,4] := 262.5288;
   DATA[1054,5] := 8.461164;
   DATA[1054,6] := 316.201;
   DATA[1054,8] := 1.0;
   DATA[1054,9] := 1.0;
   DATA[1054,10] := 1.0;
   DATA[1054,11] := 2.000768;
   DATA[1054,13] := 1011.119;
   DATA[1054,14] := 1.0;
   DATA[1054,15] := 1.0;
   DATA[1054,16] := 1.0;
   DATA[1054,17] := 1.0;
   DATA[1054,18] := 1.0;
   DATA[1054,19] := 1.0;
   DATA[1054,20] := 148.808;
   DATA[1054,21] := 154.8321;
   DATA[1054,22] := 1.712748;
   DATA[1054,23] := 891.7714;
   DATA[1054,24] := 2.0;
   DATA[1054,25] := 2.0;
   DATA[1054,26] := 7.87798;
   DATA[1054,27] := 143.9375;
   DATA[1054,28] := 263.1056;
   DATA[1054,29] := 12.03538;
   DATA[1054,30] := 1.724173;
   DATA[1054,31] := 1.293967;
   DATA[1054,32] := 0.7353967;
   DATA[1054,33] := 0.3081062;
   DATA[1054,34] := 2.0;
   DATA[1054,35] := 250.0961;
   DATA[1054,36] := 1.665972;
   DATA[1054,37] := 188.9259;
   DATA[1054,38] := 0.000128152;
   DATA[1054,39] := 1.0;
   DATA[1055,0] := 2.540115;
   DATA[1055,1] := 682.527;
   DATA[1055,2] := 2.0;
   DATA[1055,3] := 1.0;
   DATA[1055,4] := 262.5288;
   DATA[1055,5] := 8.46533;
   DATA[1055,6] := 316.201;
   DATA[1055,8] := 1.0;
   DATA[1055,9] := 1.0;
   DATA[1055,10] := 1.0;
   DATA[1055,11] := 2.000768;
   DATA[1055,13] := 1011.039;
   DATA[1055,14] := 1.0;
   DATA[1055,15] := 1.0;
   DATA[1055,16] := 1.0;
   DATA[1055,17] := 1.0;
   DATA[1055,18] := 1.0;
   DATA[1055,19] := 1.0;
   DATA[1055,20] := 148.808;
   DATA[1055,21] := 154.8321;
   DATA[1055,22] := 1.712748;
   DATA[1055,23] := 890.9639;
   DATA[1055,24] := 2.0;
   DATA[1055,25] := 2.0;
   DATA[1055,26] := 7.87798;
   DATA[1055,27] := 143.9375;
   DATA[1055,28] := 263.1056;
   DATA[1055,29] := 12.03538;
   DATA[1055,30] := 1.723532;
   DATA[1055,31] := 1.30178;
   DATA[1055,32] := 0.7353967;
   DATA[1055,33] := 0.3082983;
   DATA[1055,34] := 2.0;
   DATA[1055,35] := 250.0801;
   DATA[1055,36] := 1.665972;
   DATA[1055,37] := 188.9259;
   DATA[1055,38] := 0.000128152;
   DATA[1055,39] := 1.0;
   DATA[1056,0] := 2.542677;
   DATA[1056,1] := 682.8802;
   DATA[1056,2] := 2.0;
   DATA[1056,3] := 1.0;
   DATA[1056,4] := 262.5288;
   DATA[1056,5] := 8.46533;
   DATA[1056,6] := 316.201;
   DATA[1056,8] := 1.0;
   DATA[1056,9] := 1.0;
   DATA[1056,10] := 1.0;
   DATA[1056,11] := 2.000768;
   DATA[1056,13] := 1011.119;
   DATA[1056,14] := 1.0;
   DATA[1056,15] := 1.0;
   DATA[1056,16] := 1.0;
   DATA[1056,17] := 1.0;
   DATA[1056,18] := 1.0;
   DATA[1056,19] := 1.0;
   DATA[1056,20] := 148.808;
   DATA[1056,21] := 154.8321;
   DATA[1056,22] := 1.712363;
   DATA[1056,23] := 891.0792;
   DATA[1056,24] := 2.0;
   DATA[1056,25] := 2.0;
   DATA[1056,26] := 7.87798;
   DATA[1056,27] := 143.9375;
   DATA[1056,28] := 263.1056;
   DATA[1056,29] := 12.03538;
   DATA[1056,30] := 1.723532;
   DATA[1056,31] := 1.30178;
   DATA[1056,32] := 0.7353967;
   DATA[1056,33] := 0.3082983;
   DATA[1056,34] := 2.0;
   DATA[1056,35] := 250.0801;
   DATA[1056,36] := 1.665972;
   DATA[1056,37] := 188.9259;
   DATA[1056,38] := 0.000128152;
   DATA[1056,39] := 1.0;
   DATA[1057,0] := 2.542677;
   DATA[1057,1] := 682.8802;
   DATA[1057,2] := 2.0;
   DATA[1057,3] := 1.0;
   DATA[1057,4] := 262.5288;
   DATA[1057,5] := 8.46533;
   DATA[1057,6] := 316.201;
   DATA[1057,8] := 1.0;
   DATA[1057,9] := 1.0;
   DATA[1057,10] := 1.0;
   DATA[1057,11] := 2.000768;
   DATA[1057,13] := 1011.119;
   DATA[1057,14] := 1.0;
   DATA[1057,15] := 1.0;
   DATA[1057,16] := 1.0;
   DATA[1057,17] := 1.0;
   DATA[1057,18] := 1.0;
   DATA[1057,19] := 1.0;
   DATA[1057,20] := 148.808;
   DATA[1057,21] := 154.8321;
   DATA[1057,22] := 1.712363;
   DATA[1057,23] := 891.0792;
   DATA[1057,24] := 2.0;
   DATA[1057,25] := 2.0;
   DATA[1057,26] := 7.87798;
   DATA[1057,27] := 143.9375;
   DATA[1057,28] := 263.1056;
   DATA[1057,29] := 12.03538;
   DATA[1057,30] := 1.723532;
   DATA[1057,31] := 1.30178;
   DATA[1057,32] := 0.7353967;
   DATA[1057,33] := 0.3082983;
   DATA[1057,34] := 2.0;
   DATA[1057,35] := 250.0801;
   DATA[1057,36] := 1.665972;
   DATA[1057,37] := 188.9259;
   DATA[1057,38] := 0.000128152;
   DATA[1057,39] := 1.0;
   DATA[1058,0] := 2.548121;
   DATA[1058,1] := 683.469;
   DATA[1058,2] := 2.0;
   DATA[1058,3] := 1.0;
   DATA[1058,4] := 262.5288;
   DATA[1058,5] := 8.46533;
   DATA[1058,6] := 316.201;
   DATA[1058,8] := 1.0;
   DATA[1058,9] := 1.0;
   DATA[1058,10] := 1.0;
   DATA[1058,11] := 2.000768;
   DATA[1058,13] := 1010.839;
   DATA[1058,14] := 1.0;
   DATA[1058,15] := 1.0;
   DATA[1058,16] := 1.0;
   DATA[1058,17] := 1.0;
   DATA[1058,18] := 1.0;
   DATA[1058,19] := 1.0;
   DATA[1058,20] := 148.808;
   DATA[1058,21] := 154.8321;
   DATA[1058,22] := 1.712235;
   DATA[1058,23] := 890.9254;
   DATA[1058,24] := 2.0;
   DATA[1058,25] := 2.0;
   DATA[1058,26] := 7.87798;
   DATA[1058,27] := 143.9375;
   DATA[1058,28] := 263.1056;
   DATA[1058,29] := 12.03538;
   DATA[1058,30] := 1.72443;
   DATA[1058,31] := 1.285769;
   DATA[1058,32] := 0.7353967;
   DATA[1058,33] := 0.3082983;
   DATA[1058,34] := 2.0;
   DATA[1058,35] := 250.0801;
   DATA[1058,36] := 1.665972;
   DATA[1058,37] := 189.0541;
   DATA[1058,38] := 0.000128152;
   DATA[1058,39] := 1.0;
   DATA[1059,0] := 2.550684;
   DATA[1059,1] := 683.783;
   DATA[1059,2] := 2.0;
   DATA[1059,3] := 1.0;
   DATA[1059,4] := 262.5288;
   DATA[1059,5] := 8.466612;
   DATA[1059,6] := 316.2779;
   DATA[1059,8] := 1.0;
   DATA[1059,9] := 1.0;
   DATA[1059,10] := 1.0;
   DATA[1059,11] := 2.000768;
   DATA[1059,13] := 1010.879;
   DATA[1059,14] := 1.0;
   DATA[1059,15] := 1.0;
   DATA[1059,16] := 1.0;
   DATA[1059,17] := 1.0;
   DATA[1059,18] := 1.0;
   DATA[1059,19] := 1.0;
   DATA[1059,20] := 148.808;
   DATA[1059,21] := 154.8321;
   DATA[1059,22] := 1.712235;
   DATA[1059,23] := 890.9254;
   DATA[1059,24] := 2.0;
   DATA[1059,25] := 2.0;
   DATA[1059,26] := 7.87798;
   DATA[1059,27] := 143.9375;
   DATA[1059,28] := 263.1056;
   DATA[1059,29] := 12.03538;
   DATA[1059,30] := 1.724686;
   DATA[1059,31] := 1.274753;
   DATA[1059,32] := 0.7353967;
   DATA[1059,33] := 0.3082983;
   DATA[1059,34] := 2.0;
   DATA[1059,35] := 250.1762;
   DATA[1059,36] := 1.665972;
   DATA[1059,37] := 189.1022;
   DATA[1059,38] := 0.000128152;
   DATA[1059,39] := 1.0;
   DATA[1060,0] := 2.550684;
   DATA[1060,1] := 683.783;
   DATA[1060,2] := 2.0;
   DATA[1060,3] := 1.0;
   DATA[1060,4] := 262.5288;
   DATA[1060,5] := 8.467573;
   DATA[1060,6] := 316.2779;
   DATA[1060,8] := 1.0;
   DATA[1060,9] := 1.0;
   DATA[1060,10] := 1.0;
   DATA[1060,11] := 2.000768;
   DATA[1060,13] := 1010.678;
   DATA[1060,14] := 1.0;
   DATA[1060,15] := 1.0;
   DATA[1060,16] := 1.0;
   DATA[1060,17] := 1.0;
   DATA[1060,18] := 1.0;
   DATA[1060,19] := 1.0;
   DATA[1060,20] := 148.808;
   DATA[1060,21] := 154.8321;
   DATA[1060,22] := 1.714926;
   DATA[1060,23] := 890.5409;
   DATA[1060,24] := 2.0;
   DATA[1060,25] := 2.0;
   DATA[1060,26] := 7.87798;
   DATA[1060,27] := 143.9375;
   DATA[1060,28] := 263.1056;
   DATA[1060,29] := 12.03538;
   DATA[1060,30] := 1.725327;
   DATA[1060,31] := 1.28103;
   DATA[1060,32] := 0.7353967;
   DATA[1060,33] := 0.3082983;
   DATA[1060,34] := 2.0;
   DATA[1060,35] := 250.3044;
   DATA[1060,36] := 1.665972;
   DATA[1060,37] := 189.1662;
   DATA[1060,38] := 0.000128152;
   DATA[1060,39] := 1.0;
   DATA[1061,0] := 2.550684;
   DATA[1061,1] := 684.0578;
   DATA[1061,2] := 2.0;
   DATA[1061,3] := 1.0;
   DATA[1061,4] := 262.5288;
   DATA[1061,5] := 8.469175;
   DATA[1061,6] := 316.2779;
   DATA[1061,8] := 1.0;
   DATA[1061,9] := 1.0;
   DATA[1061,10] := 1.0;
   DATA[1061,11] := 2.000768;
   DATA[1061,13] := 1011.079;
   DATA[1061,14] := 1.0;
   DATA[1061,15] := 1.0;
   DATA[1061,16] := 1.0;
   DATA[1061,17] := 1.0;
   DATA[1061,18] := 1.0;
   DATA[1061,19] := 1.0;
   DATA[1061,20] := 148.808;
   DATA[1061,21] := 154.8321;
   DATA[1061,22] := 1.71608;
   DATA[1061,23] := 890.3871;
   DATA[1061,24] := 2.0;
   DATA[1061,25] := 2.0;
   DATA[1061,26] := 7.87798;
   DATA[1061,27] := 143.9375;
   DATA[1061,28] := 263.1056;
   DATA[1061,29] := 12.03538;
   DATA[1061,30] := 1.725327;
   DATA[1061,31] := 1.287947;
   DATA[1061,32] := 0.7353967;
   DATA[1061,33] := 0.3082983;
   DATA[1061,34] := 2.0;
   DATA[1061,35] := 250.3044;
   DATA[1061,36] := 1.665972;
   DATA[1061,37] := 189.3265;
   DATA[1061,38] := 0.000128152;
   DATA[1061,39] := 1.0;
   DATA[1062,0] := 2.550684;
   DATA[1062,1] := 684.3326;
   DATA[1062,2] := 2.0;
   DATA[1062,3] := 1.0;
   DATA[1062,4] := 262.5288;
   DATA[1062,5] := 8.469175;
   DATA[1062,6] := 316.2779;
   DATA[1062,8] := 1.0;
   DATA[1062,9] := 1.0;
   DATA[1062,10] := 1.0;
   DATA[1062,11] := 2.000768;
   DATA[1062,13] := 1011.119;
   DATA[1062,14] := 1.0;
   DATA[1062,15] := 1.0;
   DATA[1062,16] := 1.0;
   DATA[1062,17] := 1.0;
   DATA[1062,18] := 1.0;
   DATA[1062,19] := 1.0;
   DATA[1062,20] := 148.808;
   DATA[1062,21] := 154.8321;
   DATA[1062,22] := 1.716849;
   DATA[1062,23] := 889.9257;
   DATA[1062,24] := 2.0;
   DATA[1062,25] := 2.0;
   DATA[1062,26] := 7.87798;
   DATA[1062,27] := 143.9375;
   DATA[1062,28] := 263.1056;
   DATA[1062,29] := 12.03538;
   DATA[1062,30] := 1.727634;
   DATA[1062,31] := 1.291533;
   DATA[1062,32] := 0.7353967;
   DATA[1062,33] := 0.3082983;
   DATA[1062,34] := 2.0;
   DATA[1062,35] := 250.3044;
   DATA[1062,36] := 1.665972;
   DATA[1062,37] := 189.3265;
   DATA[1062,38] := 0.000128152;
   DATA[1062,39] := 1.0;
   DATA[1063,0] := 2.553566;
   DATA[1063,1] := 685.0391;
   DATA[1063,2] := 2.0;
   DATA[1063,3] := 1.0;
   DATA[1063,4] := 262.5288;
   DATA[1063,5] := 8.469175;
   DATA[1063,6] := 316.2779;
   DATA[1063,8] := 1.0;
   DATA[1063,9] := 1.0;
   DATA[1063,10] := 1.0;
   DATA[1063,11] := 2.000768;
   DATA[1063,13] := 1011.079;
   DATA[1063,14] := 1.0;
   DATA[1063,15] := 1.0;
   DATA[1063,16] := 1.0;
   DATA[1063,17] := 1.0;
   DATA[1063,18] := 1.0;
   DATA[1063,19] := 1.0;
   DATA[1063,20] := 148.808;
   DATA[1063,21] := 154.8321;
   DATA[1063,22] := 1.717489;
   DATA[1063,23] := 889.5796;
   DATA[1063,24] := 2.0;
   DATA[1063,25] := 2.0;
   DATA[1063,26] := 7.87798;
   DATA[1063,27] := 143.8349;
   DATA[1063,28] := 263.1056;
   DATA[1063,29] := 12.03538;
   DATA[1063,30] := 1.72789;
   DATA[1063,31] := 1.292174;
   DATA[1063,32] := 0.7353967;
   DATA[1063,33] := 0.3082983;
   DATA[1063,34] := 2.0;
   DATA[1063,35] := 250.3044;
   DATA[1063,36] := 1.665972;
   DATA[1063,37] := 189.3265;
   DATA[1063,38] := 0.000128152;
   DATA[1063,39] := 1.0;
   DATA[1064,0] := 2.553566;
   DATA[1064,1] := 685.5494;
   DATA[1064,2] := 2.0;
   DATA[1064,3] := 1.0;
   DATA[1064,4] := 262.5288;
   DATA[1064,5] := 8.469175;
   DATA[1064,6] := 316.2779;
   DATA[1064,8] := 1.0;
   DATA[1064,9] := 1.0;
   DATA[1064,10] := 1.0;
   DATA[1064,11] := 2.000768;
   DATA[1064,13] := 1010.919;
   DATA[1064,14] := 1.0;
   DATA[1064,15] := 1.0;
   DATA[1064,16] := 1.0;
   DATA[1064,17] := 1.0;
   DATA[1064,18] := 1.0;
   DATA[1064,19] := 1.0;
   DATA[1064,20] := 148.808;
   DATA[1064,21] := 154.8321;
   DATA[1064,22] := 1.717489;
   DATA[1064,23] := 889.4258;
   DATA[1064,24] := 2.0;
   DATA[1064,25] := 2.0;
   DATA[1064,26] := 7.87798;
   DATA[1064,27] := 143.8349;
   DATA[1064,28] := 263.1056;
   DATA[1064,29] := 12.03538;
   DATA[1064,30] := 1.72789;
   DATA[1064,31] := 1.277443;
   DATA[1064,32] := 0.7353967;
   DATA[1064,33] := 0.3075937;
   DATA[1064,34] := 2.0;
   DATA[1064,35] := 250.3044;
   DATA[1064,36] := 1.665972;
   DATA[1064,37] := 189.3265;
   DATA[1064,38] := 0.000128152;
   DATA[1064,39] := 1.0;
   DATA[1065,0] := 2.54652;
   DATA[1065,1] := 685.942;
   DATA[1065,2] := 2.0;
   DATA[1065,3] := 1.0;
   DATA[1065,4] := 262.5288;
   DATA[1065,5] := 8.469175;
   DATA[1065,6] := 316.2779;
   DATA[1065,8] := 1.0;
   DATA[1065,9] := 1.0;
   DATA[1065,10] := 1.0;
   DATA[1065,11] := 2.000768;
   DATA[1065,13] := 1011.039;
   DATA[1065,14] := 1.0;
   DATA[1065,15] := 1.0;
   DATA[1065,16] := 1.0;
   DATA[1065,17] := 1.0;
   DATA[1065,18] := 1.0;
   DATA[1065,19] := 1.0;
   DATA[1065,20] := 148.808;
   DATA[1065,21] := 154.8321;
   DATA[1065,22] := 1.717489;
   DATA[1065,23] := 888.849;
   DATA[1065,24] := 2.0;
   DATA[1065,25] := 2.0;
   DATA[1065,26] := 7.87798;
   DATA[1065,27] := 143.8349;
   DATA[1065,28] := 263.1056;
   DATA[1065,29] := 12.03538;
   DATA[1065,30] := 1.725583;
   DATA[1065,31] := 1.261816;
   DATA[1065,32] := 0.7353967;
   DATA[1065,33] := 0.306761;
   DATA[1065,34] := 2.0;
   DATA[1065,35] := 250.4005;
   DATA[1065,36] := 1.665972;
   DATA[1065,37] := 189.3265;
   DATA[1065,38] := 0.000128152;
   DATA[1065,39] := 1.0;
   DATA[1066,0] := 2.54652;
   DATA[1066,1] := 686.4915;
   DATA[1066,2] := 2.0;
   DATA[1066,3] := 1.0;
   DATA[1066,4] := 262.5288;
   DATA[1066,5] := 8.469175;
   DATA[1066,6] := 316.2779;
   DATA[1066,8] := 1.0;
   DATA[1066,9] := 1.0;
   DATA[1066,10] := 1.0;
   DATA[1066,11] := 2.000768;
   DATA[1066,13] := 1010.558;
   DATA[1066,14] := 1.0;
   DATA[1066,15] := 1.0;
   DATA[1066,16] := 1.0;
   DATA[1066,17] := 1.0;
   DATA[1066,18] := 1.0;
   DATA[1066,19] := 1.0;
   DATA[1066,20] := 148.808;
   DATA[1066,21] := 154.8321;
   DATA[1066,22] := 1.717489;
   DATA[1066,23] := 888.6952;
   DATA[1066,24] := 2.0;
   DATA[1066,25] := 2.0;
   DATA[1066,26] := 7.87798;
   DATA[1066,27] := 143.8349;
   DATA[1066,28] := 263.1056;
   DATA[1066,29] := 12.22763;
   DATA[1066,30] := 1.72507;
   DATA[1066,31] := 1.261816;
   DATA[1066,32] := 0.7353967;
   DATA[1066,33] := 0.3065048;
   DATA[1066,34] := 2.0;
   DATA[1066,35] := 250.4005;
   DATA[1066,36] := 1.665972;
   DATA[1066,37] := 189.2624;
   DATA[1066,38] := 0.000128152;
   DATA[1066,39] := 1.0;
   DATA[1067,0] := 2.551965;
   DATA[1067,1] := 687.041;
   DATA[1067,2] := 2.0;
   DATA[1067,3] := 1.0;
   DATA[1067,4] := 262.5288;
   DATA[1067,5] := 8.466932;
   DATA[1067,6] := 316.2779;
   DATA[1067,8] := 1.0;
   DATA[1067,9] := 1.0;
   DATA[1067,10] := 1.0;
   DATA[1067,11] := 2.000768;
   DATA[1067,13] := 1011.039;
   DATA[1067,14] := 1.0;
   DATA[1067,15] := 1.0;
   DATA[1067,16] := 1.0;
   DATA[1067,17] := 1.0;
   DATA[1067,18] := 1.0;
   DATA[1067,19] := 1.0;
   DATA[1067,20] := 148.808;
   DATA[1067,21] := 154.8321;
   DATA[1067,22] := 1.717105;
   DATA[1067,23] := 888.08;
   DATA[1067,24] := 2.0;
   DATA[1067,25] := 2.0;
   DATA[1067,26] := 7.87798;
   DATA[1067,27] := 143.8349;
   DATA[1067,28] := 263.1056;
   DATA[1067,29] := 12.22763;
   DATA[1067,30] := 1.72507;
   DATA[1067,31] := 1.261816;
   DATA[1067,32] := 0.7353967;
   DATA[1067,33] := 0.3065048;
   DATA[1067,34] := 2.0;
   DATA[1067,35] := 250.4005;
   DATA[1067,36] := 1.665972;
   DATA[1067,37] := 189.2624;
   DATA[1067,38] := 0.000128152;
   DATA[1067,39] := 1.0;
   DATA[1068,0] := 2.551965;
   DATA[1068,1] := 687.2766;
   DATA[1068,2] := 2.0;
   DATA[1068,3] := 1.0;
   DATA[1068,4] := 262.5288;
   DATA[1068,5] := 8.466932;
   DATA[1068,6] := 316.2779;
   DATA[1068,8] := 1.0;
   DATA[1068,9] := 1.0;
   DATA[1068,10] := 1.0;
   DATA[1068,11] := 2.000768;
   DATA[1068,13] := 1010.839;
   DATA[1068,14] := 1.0;
   DATA[1068,15] := 1.0;
   DATA[1068,16] := 1.0;
   DATA[1068,17] := 1.0;
   DATA[1068,18] := 1.0;
   DATA[1068,19] := 1.0;
   DATA[1068,20] := 148.808;
   DATA[1068,21] := 154.8321;
   DATA[1068,22] := 1.715439;
   DATA[1068,23] := 887.8877;
   DATA[1068,24] := 2.0;
   DATA[1068,25] := 2.0;
   DATA[1068,26] := 7.87798;
   DATA[1068,27] := 143.8349;
   DATA[1068,28] := 263.1056;
   DATA[1068,29] := 12.22763;
   DATA[1068,30] := 1.72507;
   DATA[1068,31] := 1.277059;
   DATA[1068,32] := 0.7353967;
   DATA[1068,33] := 0.3065048;
   DATA[1068,34] := 2.0;
   DATA[1068,35] := 250.4005;
   DATA[1068,36] := 1.665972;
   DATA[1068,37] := 189.2624;
   DATA[1068,38] := 0.000128152;
   DATA[1068,39] := 1.0;
   DATA[1069,0] := 2.551965;
   DATA[1069,1] := 687.6691;
   DATA[1069,2] := 2.0;
   DATA[1069,3] := 1.0;
   DATA[1069,4] := 262.5288;
   DATA[1069,5] := 8.466932;
   DATA[1069,6] := 316.2779;
   DATA[1069,8] := 1.0;
   DATA[1069,9] := 1.0;
   DATA[1069,10] := 1.0;
   DATA[1069,11] := 2.000768;
   DATA[1069,13] := 1010.959;
   DATA[1069,14] := 1.0;
   DATA[1069,15] := 1.0;
   DATA[1069,16] := 1.0;
   DATA[1069,17] := 1.0;
   DATA[1069,18] := 1.0;
   DATA[1069,19] := 1.0;
   DATA[1069,20] := 148.808;
   DATA[1069,21] := 154.8321;
   DATA[1069,22] := 1.715439;
   DATA[1069,23] := 887.6185;
   DATA[1069,24] := 2.0;
   DATA[1069,25] := 2.0;
   DATA[1069,26] := 7.87798;
   DATA[1069,27] := 143.8349;
   DATA[1069,28] := 263.1056;
   DATA[1069,29] := 12.22763;
   DATA[1069,30] := 1.72507;
   DATA[1069,31] := 1.297169;
   DATA[1069,32] := 0.7353967;
   DATA[1069,33] := 0.3065048;
   DATA[1069,34] := 2.0;
   DATA[1069,35] := 250.4005;
   DATA[1069,36] := 1.665972;
   DATA[1069,37] := 189.2624;
   DATA[1069,38] := 0.000128152;
   DATA[1069,39] := 1.0;
   DATA[1070,0] := 2.550043;
   DATA[1070,1] := 688.2186;
   DATA[1070,2] := 2.0;
   DATA[1070,3] := 1.0;
   DATA[1070,4] := 262.5288;
   DATA[1070,5] := 8.466932;
   DATA[1070,6] := 316.2779;
   DATA[1070,8] := 1.0;
   DATA[1070,9] := 1.0;
   DATA[1070,10] := 1.0;
   DATA[1070,11] := 2.000768;
   DATA[1070,13] := 1010.678;
   DATA[1070,14] := 1.0;
   DATA[1070,15] := 1.0;
   DATA[1070,16] := 1.0;
   DATA[1070,17] := 1.0;
   DATA[1070,18] := 1.0;
   DATA[1070,19] := 1.0;
   DATA[1070,20] := 148.808;
   DATA[1070,21] := 154.8321;
   DATA[1070,22] := 1.715439;
   DATA[1070,23] := 887.0418;
   DATA[1070,24] := 2.0;
   DATA[1070,25] := 2.0;
   DATA[1070,26] := 7.87798;
   DATA[1070,27] := 143.8349;
   DATA[1070,28] := 263.1056;
   DATA[1070,29] := 12.22763;
   DATA[1070,30] := 1.726865;
   DATA[1070,31] := 1.302165;
   DATA[1070,32] := 0.7353967;
   DATA[1070,33] := 0.3065048;
   DATA[1070,34] := 2.0;
   DATA[1070,35] := 250.4005;
   DATA[1070,36] := 1.665972;
   DATA[1070,37] := 189.2464;
   DATA[1070,38] := 0.000128152;
   DATA[1070,39] := 1.0;
   DATA[1071,0] := 2.543958;
   DATA[1071,1] := 688.6896;
   DATA[1071,2] := 2.0;
   DATA[1071,3] := 1.0;
   DATA[1071,4] := 262.5288;
   DATA[1071,5] := 8.467573;
   DATA[1071,6] := 316.2779;
   DATA[1071,8] := 1.0;
   DATA[1071,9] := 1.0;
   DATA[1071,10] := 1.0;
   DATA[1071,11] := 2.000768;
   DATA[1071,13] := 1010.919;
   DATA[1071,14] := 1.0;
   DATA[1071,15] := 1.0;
   DATA[1071,16] := 1.0;
   DATA[1071,17] := 1.0;
   DATA[1071,18] := 1.0;
   DATA[1071,19] := 1.0;
   DATA[1071,20] := 148.808;
   DATA[1071,21] := 154.8321;
   DATA[1071,22] := 1.715439;
   DATA[1071,23] := 886.9649;
   DATA[1071,24] := 2.0;
   DATA[1071,25] := 2.0;
   DATA[1071,26] := 7.87798;
   DATA[1071,27] := 143.8349;
   DATA[1071,28] := 263.1056;
   DATA[1071,29] := 12.22763;
   DATA[1071,30] := 1.726865;
   DATA[1071,31] := 1.302165;
   DATA[1071,32] := 0.7353967;
   DATA[1071,33] := 0.3065048;
   DATA[1071,34] := 2.0;
   DATA[1071,35] := 250.4005;
   DATA[1071,36] := 1.665972;
   DATA[1071,37] := 189.2464;
   DATA[1071,38] := 0.000128152;
   DATA[1071,39] := 1.0;
   DATA[1072,0] := 2.543958;
   DATA[1072,1] := 689.2392;
   DATA[1072,2] := 2.0;
   DATA[1072,3] := 1.0;
   DATA[1072,4] := 262.5288;
   DATA[1072,5] := 8.468855;
   DATA[1072,6] := 316.3804;
   DATA[1072,8] := 1.0;
   DATA[1072,9] := 1.0;
   DATA[1072,10] := 1.0;
   DATA[1072,11] := 2.000768;
   DATA[1072,13] := 1010.959;
   DATA[1072,14] := 1.0;
   DATA[1072,15] := 1.0;
   DATA[1072,16] := 1.0;
   DATA[1072,17] := 1.0;
   DATA[1072,18] := 1.0;
   DATA[1072,19] := 1.0;
   DATA[1072,20] := 148.808;
   DATA[1072,21] := 154.8321;
   DATA[1072,22] := 1.715439;
   DATA[1072,23] := 886.5419;
   DATA[1072,24] := 2.0;
   DATA[1072,25] := 2.0;
   DATA[1072,26] := 7.87798;
   DATA[1072,27] := 143.8349;
   DATA[1072,28] := 263.1056;
   DATA[1072,29] := 12.07383;
   DATA[1072,30] := 1.726865;
   DATA[1072,31] := 1.301652;
   DATA[1072,32] := 0.7353967;
   DATA[1072,33] := 0.3065048;
   DATA[1072,34] := 2.0;
   DATA[1072,35] := 250.4005;
   DATA[1072,36] := 1.665972;
   DATA[1072,37] := 189.2464;
   DATA[1072,38] := 0.000128152;
   DATA[1072,39] := 1.0;
   DATA[1073,0] := 2.540435;
   DATA[1073,1] := 689.9457;
   DATA[1073,2] := 2.0;
   DATA[1073,3] := 1.0;
   DATA[1073,4] := 262.5288;
   DATA[1073,5] := 8.468855;
   DATA[1073,6] := 316.3804;
   DATA[1073,8] := 1.0;
   DATA[1073,9] := 1.0;
   DATA[1073,10] := 1.0;
   DATA[1073,11] := 2.000768;
   DATA[1073,13] := 1010.959;
   DATA[1073,14] := 1.0;
   DATA[1073,15] := 1.0;
   DATA[1073,16] := 1.0;
   DATA[1073,17] := 1.0;
   DATA[1073,18] := 1.0;
   DATA[1073,19] := 1.0;
   DATA[1073,20] := 148.808;
   DATA[1073,21] := 154.8321;
   DATA[1073,22] := 1.715439;
   DATA[1073,23] := 886.5804;
   DATA[1073,24] := 2.0;
   DATA[1073,25] := 2.0;
   DATA[1073,26] := 7.87798;
   DATA[1073,27] := 143.8349;
   DATA[1073,28] := 263.1056;
   DATA[1073,29] := 12.07383;
   DATA[1073,30] := 1.726865;
   DATA[1073,31] := 1.284873;
   DATA[1073,32] := 0.7353967;
   DATA[1073,33] := 0.3081703;
   DATA[1073,34] := 2.0;
   DATA[1073,35] := 250.4005;
   DATA[1073,36] := 1.665972;
   DATA[1073,37] := 189.2464;
   DATA[1073,38] := 0.000128152;
   DATA[1073,39] := 1.0;
   DATA[1074,0] := 2.533709;
   DATA[1074,1] := 690.0635;
   DATA[1074,2] := 2.0;
   DATA[1074,3] := 1.0;
   DATA[1074,4] := 262.5288;
   DATA[1074,5] := 8.468855;
   DATA[1074,6] := 316.3804;
   DATA[1074,8] := 1.0;
   DATA[1074,9] := 1.0;
   DATA[1074,10] := 1.0;
   DATA[1074,11] := 2.000768;
   DATA[1074,13] := 1011.079;
   DATA[1074,14] := 1.0;
   DATA[1074,15] := 1.0;
   DATA[1074,16] := 1.0;
   DATA[1074,17] := 1.0;
   DATA[1074,18] := 1.0;
   DATA[1074,19] := 1.0;
   DATA[1074,20] := 148.808;
   DATA[1074,21] := 154.8321;
   DATA[1074,22] := 1.715439;
   DATA[1074,23] := 886.0036;
   DATA[1074,24] := 2.0;
   DATA[1074,25] := 2.0;
   DATA[1074,26] := 7.87798;
   DATA[1074,27] := 143.8349;
   DATA[1074,28] := 263.1056;
   DATA[1074,29] := 12.07383;
   DATA[1074,30] := 1.726865;
   DATA[1074,31] := 1.282311;
   DATA[1074,32] := 0.7353967;
   DATA[1074,33] := 0.3081703;
   DATA[1074,34] := 2.0;
   DATA[1074,35] := 250.4005;
   DATA[1074,36] := 1.730048;
   DATA[1074,37] := 189.2464;
   DATA[1074,38] := 0.000128152;
   DATA[1074,39] := 1.0;
   DATA[1075,0] := 2.529225;
   DATA[1075,1] := 690.7308;
   DATA[1075,2] := 2.0;
   DATA[1075,3] := 1.0;
   DATA[1075,4] := 262.5288;
   DATA[1075,5] := 8.466932;
   DATA[1075,6] := 316.3804;
   DATA[1075,8] := 1.0;
   DATA[1075,9] := 1.0;
   DATA[1075,10] := 1.0;
   DATA[1075,11] := 2.010372;
   DATA[1075,13] := 1011.039;
   DATA[1075,14] := 1.0;
   DATA[1075,15] := 1.0;
   DATA[1075,16] := 1.0;
   DATA[1075,17] := 1.0;
   DATA[1075,18] := 1.0;
   DATA[1075,19] := 1.0;
   DATA[1075,20] := 148.808;
   DATA[1075,21] := 154.8321;
   DATA[1075,22] := 1.715439;
   DATA[1075,23] := 885.8882;
   DATA[1075,24] := 2.0;
   DATA[1075,25] := 2.0;
   DATA[1075,26] := 7.87798;
   DATA[1075,27] := 143.8349;
   DATA[1075,28] := 263.1056;
   DATA[1075,29] := 12.07383;
   DATA[1075,30] := 1.726865;
   DATA[1075,31] := 1.286666;
   DATA[1075,32] := 0.7353967;
   DATA[1075,33] := 0.3081703;
   DATA[1075,34] := 2.0;
   DATA[1075,35] := 250.5447;
   DATA[1075,36] := 1.730048;
   DATA[1075,37] := 189.2464;
   DATA[1075,38] := 0.000128152;
   DATA[1075,39] := 1.0;
   DATA[1076,0] := 2.529225;
   DATA[1076,1] := 691.2411;
   DATA[1076,2] := 2.0;
   DATA[1076,3] := 1.0;
   DATA[1076,4] := 262.5288;
   DATA[1076,5] := 8.464369;
   DATA[1076,6] := 316.3804;
   DATA[1076,8] := 1.0;
   DATA[1076,9] := 1.0;
   DATA[1076,10] := 1.0;
   DATA[1076,11] := 2.010372;
   DATA[1076,13] := 1011.079;
   DATA[1076,14] := 1.0;
   DATA[1076,15] := 1.0;
   DATA[1076,16] := 1.0;
   DATA[1076,17] := 1.0;
   DATA[1076,18] := 1.0;
   DATA[1076,19] := 1.0;
   DATA[1076,20] := 148.808;
   DATA[1076,21] := 154.8321;
   DATA[1076,22] := 1.715439;
   DATA[1076,23] := 885.6191;
   DATA[1076,24] := 2.0;
   DATA[1076,25] := 2.0;
   DATA[1076,26] := 7.87798;
   DATA[1076,27] := 143.8349;
   DATA[1076,28] := 263.1056;
   DATA[1076,29] := 12.07383;
   DATA[1076,30] := 1.726865;
   DATA[1076,31] := 1.281798;
   DATA[1076,32] := 0.7353967;
   DATA[1076,33] := 0.3081703;
   DATA[1076,34] := 2.0;
   DATA[1076,35] := 250.5447;
   DATA[1076,36] := 1.730048;
   DATA[1076,37] := 189.2464;
   DATA[1076,38] := 0.000128152;
   DATA[1076,39] := 1.0;
   DATA[1077,0] := 2.543638;
   DATA[1077,1] := 691.5944;
   DATA[1077,2] := 2.0;
   DATA[1077,3] := 1.0;
   DATA[1077,4] := 262.5288;
   DATA[1077,5] := 8.464369;
   DATA[1077,6] := 316.3804;
   DATA[1077,8] := 1.0;
   DATA[1077,9] := 1.0;
   DATA[1077,10] := 1.0;
   DATA[1077,11] := 2.010372;
   DATA[1077,13] := 1010.718;
   DATA[1077,14] := 1.0;
   DATA[1077,15] := 1.0;
   DATA[1077,16] := 1.0;
   DATA[1077,17] := 1.0;
   DATA[1077,18] := 1.0;
   DATA[1077,19] := 1.0;
   DATA[1077,20] := 148.808;
   DATA[1077,21] := 154.8321;
   DATA[1077,22] := 1.715439;
   DATA[1077,23] := 885.0038;
   DATA[1077,24] := 2.0;
   DATA[1077,25] := 2.0;
   DATA[1077,26] := 7.87798;
   DATA[1077,27] := 143.8349;
   DATA[1077,28] := 263.1056;
   DATA[1077,29] := 12.07383;
   DATA[1077,30] := 1.726352;
   DATA[1077,31] := 1.28167;
   DATA[1077,32] := 0.7353967;
   DATA[1077,33] := 0.3081703;
   DATA[1077,34] := 2.0;
   DATA[1077,35] := 250.5447;
   DATA[1077,36] := 1.730048;
   DATA[1077,37] := 189.2464;
   DATA[1077,38] := 0.000128152;
   DATA[1077,39] := 1.0;
   DATA[1078,0] := 2.549082;
   DATA[1078,1] := 692.3401;
   DATA[1078,2] := 2.0;
   DATA[1078,3] := 1.0;
   DATA[1078,4] := 262.5288;
   DATA[1078,5] := 8.464369;
   DATA[1078,6] := 316.3804;
   DATA[1078,8] := 1.0;
   DATA[1078,9] := 1.0;
   DATA[1078,10] := 1.0;
   DATA[1078,11] := 2.010372;
   DATA[1078,13] := 1010.919;
   DATA[1078,14] := 1.0;
   DATA[1078,15] := 1.0;
   DATA[1078,16] := 1.0;
   DATA[1078,17] := 1.0;
   DATA[1078,18] := 1.0;
   DATA[1078,19] := 1.0;
   DATA[1078,20] := 148.808;
   DATA[1078,21] := 154.6526;
   DATA[1078,22] := 1.715952;
   DATA[1078,23] := 884.6578;
   DATA[1078,24] := 2.0;
   DATA[1078,25] := 2.0;
   DATA[1078,26] := 7.87798;
   DATA[1078,27] := 143.8349;
   DATA[1078,28] := 263.1056;
   DATA[1078,29] := 12.07383;
   DATA[1078,30] := 1.725968;
   DATA[1078,31] := 1.274113;
   DATA[1078,32] := 0.7353967;
   DATA[1078,33] := 0.3084905;
   DATA[1078,34] := 2.0;
   DATA[1078,35] := 250.5447;
   DATA[1078,36] := 1.730048;
   DATA[1078,37] := 189.2464;
   DATA[1078,38] := 0.000128152;
   DATA[1078,39] := 1.0;
   DATA[1079,0] := 2.550043;
   DATA[1079,1] := 692.6149;
   DATA[1079,2] := 2.0;
   DATA[1079,3] := 1.0;
   DATA[1079,4] := 262.5288;
   DATA[1079,5] := 8.464369;
   DATA[1079,6] := 316.3804;
   DATA[1079,8] := 1.0;
   DATA[1079,9] := 1.0;
   DATA[1079,10] := 1.0;
   DATA[1079,11] := 2.010372;
   DATA[1079,13] := 1010.718;
   DATA[1079,14] := 1.0;
   DATA[1079,15] := 1.0;
   DATA[1079,16] := 1.0;
   DATA[1079,17] := 1.0;
   DATA[1079,18] := 1.0;
   DATA[1079,19] := 1.0;
   DATA[1079,20] := 148.808;
   DATA[1079,21] := 154.6526;
   DATA[1079,22] := 1.715952;
   DATA[1079,23] := 884.6193;
   DATA[1079,24] := 2.0;
   DATA[1079,25] := 2.0;
   DATA[1079,26] := 7.87798;
   DATA[1079,27] := 143.8349;
   DATA[1079,28] := 263.1056;
   DATA[1079,29] := 12.07383;
   DATA[1079,30] := 1.725968;
   DATA[1079,31] := 1.272576;
   DATA[1079,32] := 0.7353967;
   DATA[1079,33] := 0.3084905;
   DATA[1079,34] := 2.0;
   DATA[1079,35] := 250.5447;
   DATA[1079,36] := 1.69801;
   DATA[1079,37] := 189.2464;
   DATA[1079,38] := 0.000128152;
   DATA[1079,39] := 1.0;
   DATA[1080,0] := 2.550043;
   DATA[1080,1] := 693.2037;
   DATA[1080,2] := 2.0;
   DATA[1080,3] := 1.0;
   DATA[1080,4] := 262.5288;
   DATA[1080,5] := 8.464369;
   DATA[1080,6] := 316.3804;
   DATA[1080,8] := 1.0;
   DATA[1080,9] := 1.0;
   DATA[1080,10] := 1.0;
   DATA[1080,11] := 2.010372;
   DATA[1080,13] := 1010.919;
   DATA[1080,14] := 1.0;
   DATA[1080,15] := 1.0;
   DATA[1080,16] := 1.0;
   DATA[1080,17] := 1.0;
   DATA[1080,18] := 1.0;
   DATA[1080,19] := 1.0;
   DATA[1080,20] := 148.808;
   DATA[1080,21] := 154.6526;
   DATA[1080,22] := 1.715952;
   DATA[1080,23] := 884.0425;
   DATA[1080,24] := 2.0;
   DATA[1080,25] := 2.0;
   DATA[1080,26] := 7.87798;
   DATA[1080,27] := 143.8349;
   DATA[1080,28] := 263.1056;
   DATA[1080,29] := 12.07383;
   DATA[1080,30] := 1.725968;
   DATA[1080,31] := 1.280517;
   DATA[1080,32] := 0.7353967;
   DATA[1080,33] := 0.3084905;
   DATA[1080,34] := 2.0;
   DATA[1080,35] := 250.3204;
   DATA[1080,36] := 1.69801;
   DATA[1080,37] := 189.2464;
   DATA[1080,38] := 0.000128152;
   DATA[1080,39] := 1.0;
   DATA[1081,0] := 2.550043;
   DATA[1081,1] := 693.871;
   DATA[1081,2] := 2.0;
   DATA[1081,3] := 1.0;
   DATA[1081,4] := 262.5288;
   DATA[1081,5] := 8.464369;
   DATA[1081,6] := 316.3804;
   DATA[1081,8] := 1.0;
   DATA[1081,9] := 1.0;
   DATA[1081,10] := 1.0;
   DATA[1081,11] := 2.010372;
   DATA[1081,13] := 1010.638;
   DATA[1081,14] := 1.0;
   DATA[1081,15] := 1.0;
   DATA[1081,16] := 1.0;
   DATA[1081,17] := 1.0;
   DATA[1081,18] := 1.0;
   DATA[1081,19] := 1.0;
   DATA[1081,20] := 148.808;
   DATA[1081,21] := 154.6526;
   DATA[1081,22] := 1.715952;
   DATA[1081,23] := 883.6196;
   DATA[1081,24] := 2.0;
   DATA[1081,25] := 2.0;
   DATA[1081,26] := 7.87798;
   DATA[1081,27] := 143.8349;
   DATA[1081,28] := 263.1056;
   DATA[1081,29] := 12.07383;
   DATA[1081,30] := 1.725968;
   DATA[1081,31] := 1.28167;
   DATA[1081,32] := 0.7353967;
   DATA[1081,33] := 0.3070813;
   DATA[1081,34] := 2.0;
   DATA[1081,35] := 250.3204;
   DATA[1081,36] := 1.69801;
   DATA[1081,37] := 189.2464;
   DATA[1081,38] := 0.000128152;
   DATA[1081,39] := 1.0;
   DATA[1082,0] := 2.550043;
   DATA[1082,1] := 694.185;
   DATA[1082,2] := 2.0;
   DATA[1082,3] := 1.0;
   DATA[1082,4] := 262.5288;
   DATA[1082,5] := 8.464369;
   DATA[1082,6] := 316.3804;
   DATA[1082,8] := 1.0;
   DATA[1082,9] := 1.0;
   DATA[1082,10] := 1.0;
   DATA[1082,11] := 2.010372;
   DATA[1082,13] := 1010.518;
   DATA[1082,14] := 1.0;
   DATA[1082,15] := 1.0;
   DATA[1082,16] := 1.0;
   DATA[1082,17] := 1.0;
   DATA[1082,18] := 1.0;
   DATA[1082,19] := 1.0;
   DATA[1082,20] := 148.808;
   DATA[1082,21] := 154.6526;
   DATA[1082,22] := 1.715952;
   DATA[1082,23] := 883.5427;
   DATA[1082,24] := 2.0;
   DATA[1082,25] := 2.0;
   DATA[1082,26] := 7.87798;
   DATA[1082,27] := 143.8349;
   DATA[1082,28] := 263.1056;
   DATA[1082,29] := 12.07383;
   DATA[1082,30] := 1.725968;
   DATA[1082,31] := 1.28167;
   DATA[1082,32] := 0.7353967;
   DATA[1082,33] := 0.3066329;
   DATA[1082,34] := 2.0;
   DATA[1082,35] := 250.3204;
   DATA[1082,36] := 1.681991;
   DATA[1082,37] := 189.2464;
   DATA[1082,38] := 0.000128152;
   DATA[1082,39] := 1.0;
   DATA[1083,0] := 2.550043;
   DATA[1083,1] := 694.6561;
   DATA[1083,2] := 2.0;
   DATA[1083,3] := 1.0;
   DATA[1083,4] := 262.5288;
   DATA[1083,5] := 8.464369;
   DATA[1083,6] := 316.3804;
   DATA[1083,8] := 1.0;
   DATA[1083,9] := 1.0;
   DATA[1083,10] := 1.0;
   DATA[1083,11] := 2.010372;
   DATA[1083,13] := 1010.478;
   DATA[1083,14] := 1.0;
   DATA[1083,15] := 1.0;
   DATA[1083,16] := 1.0;
   DATA[1083,17] := 1.0;
   DATA[1083,18] := 1.0;
   DATA[1083,19] := 1.0;
   DATA[1083,20] := 148.808;
   DATA[1083,21] := 154.6526;
   DATA[1083,22] := 1.715952;
   DATA[1083,23] := 883.1966;
   DATA[1083,24] := 2.0;
   DATA[1083,25] := 2.0;
   DATA[1083,26] := 7.87798;
   DATA[1083,27] := 143.7067;
   DATA[1083,28] := 263.1056;
   DATA[1083,29] := 12.07383;
   DATA[1083,30] := 1.725968;
   DATA[1083,31] := 1.281158;
   DATA[1083,32] := 0.7353967;
   DATA[1083,33] := 0.3083624;
   DATA[1083,34] := 2.0;
   DATA[1083,35] := 250.3204;
   DATA[1083,36] := 1.681991;
   DATA[1083,37] := 189.2464;
   DATA[1083,38] := 0.000128152;
   DATA[1083,39] := 1.0;
   DATA[1084,0] := 2.545239;
   DATA[1084,1] := 695.0878;
   DATA[1084,2] := 2.0;
   DATA[1084,3] := 1.0;
   DATA[1084,4] := 262.5288;
   DATA[1084,5] := 8.464369;
   DATA[1084,6] := 316.3804;
   DATA[1084,8] := 1.0;
   DATA[1084,9] := 1.0;
   DATA[1084,10] := 1.0;
   DATA[1084,11] := 2.010372;
   DATA[1084,13] := 1010.518;
   DATA[1084,14] := 1.0;
   DATA[1084,15] := 1.0;
   DATA[1084,16] := 1.0;
   DATA[1084,17] := 1.0;
   DATA[1084,18] := 1.0;
   DATA[1084,19] := 1.0;
   DATA[1084,20] := 148.808;
   DATA[1084,21] := 154.6526;
   DATA[1084,22] := 1.715952;
   DATA[1084,23] := 882.889;
   DATA[1084,24] := 2.0;
   DATA[1084,25] := 2.0;
   DATA[1084,26] := 7.879262;
   DATA[1084,27] := 143.7067;
   DATA[1084,28] := 263.0415;
   DATA[1084,29] := 12.07383;
   DATA[1084,30] := 1.724942;
   DATA[1084,31] := 1.271295;
   DATA[1084,32] := 0.7353967;
   DATA[1084,33] := 0.3086827;
   DATA[1084,34] := 2.0;
   DATA[1084,35] := 250.3204;
   DATA[1084,36] := 1.681991;
   DATA[1084,37] := 189.2464;
   DATA[1084,38] := 0.000128152;
   DATA[1084,39] := 1.0;
   DATA[1085,0] := 2.533068;
   DATA[1085,1] := 695.4803;
   DATA[1085,2] := 2.0;
   DATA[1085,3] := 1.0;
   DATA[1085,4] := 262.5288;
   DATA[1085,5] := 8.464369;
   DATA[1085,6] := 316.3804;
   DATA[1085,8] := 1.0;
   DATA[1085,9] := 1.0;
   DATA[1085,10] := 1.0;
   DATA[1085,11] := 2.010372;
   DATA[1085,13] := 1010.478;
   DATA[1085,14] := 1.0;
   DATA[1085,15] := 1.0;
   DATA[1085,16] := 1.0;
   DATA[1085,17] := 1.0;
   DATA[1085,18] := 1.0;
   DATA[1085,19] := 1.0;
   DATA[1085,20] := 148.808;
   DATA[1085,21] := 154.6526;
   DATA[1085,22] := 1.715952;
   DATA[1085,23] := 882.5814;
   DATA[1085,24] := 2.0;
   DATA[1085,25] := 2.0;
   DATA[1085,26] := 7.879262;
   DATA[1085,27] := 143.5529;
   DATA[1085,28] := 263.0415;
   DATA[1085,29] := 12.07383;
   DATA[1085,30] := 1.724301;
   DATA[1085,31] := 1.270911;
   DATA[1085,32] := 0.7353967;
   DATA[1085,33] := 0.3086827;
   DATA[1085,34] := 2.0;
   DATA[1085,35] := 250.3204;
   DATA[1085,36] := 1.681991;
   DATA[1085,37] := 189.2464;
   DATA[1085,38] := 0.000128152;
   DATA[1085,39] := 1.0;
   DATA[1086,0] := 2.529225;
   DATA[1086,1] := 695.8336;
   DATA[1086,2] := 2.0;
   DATA[1086,3] := 1.0;
   DATA[1086,4] := 262.5288;
   DATA[1086,5] := 8.464369;
   DATA[1086,6] := 316.3804;
   DATA[1086,8] := 1.0;
   DATA[1086,9] := 1.0;
   DATA[1086,10] := 1.0;
   DATA[1086,11] := 2.010372;
   DATA[1086,13] := 1010.558;
   DATA[1086,14] := 1.0;
   DATA[1086,15] := 1.0;
   DATA[1086,16] := 1.0;
   DATA[1086,17] := 1.0;
   DATA[1086,18] := 1.0;
   DATA[1086,19] := 1.0;
   DATA[1086,20] := 148.808;
   DATA[1086,21] := 154.6526;
   DATA[1086,22] := 1.715952;
   DATA[1086,23] := 882.12;
   DATA[1086,24] := 2.0;
   DATA[1086,25] := 2.0;
   DATA[1086,26] := 7.879262;
   DATA[1086,27] := 143.5529;
   DATA[1086,28] := 263.0095;
   DATA[1086,29] := 12.07383;
   DATA[1086,30] := 1.724045;
   DATA[1086,31] := 1.289484;
   DATA[1086,32] := 0.7353967;
   DATA[1086,33] := 0.3086827;
   DATA[1086,34] := 2.0;
   DATA[1086,35] := 250.3204;
   DATA[1086,36] := 1.681991;
   DATA[1086,37] := 189.2464;
   DATA[1086,38] := 0.000128152;
   DATA[1086,39] := 1.0;
   DATA[1087,0] := 2.529225;
   DATA[1087,1] := 696.4617;
   DATA[1087,2] := 2.0;
   DATA[1087,3] := 1.0;
   DATA[1087,4] := 262.5288;
   DATA[1087,5] := 8.464369;
   DATA[1087,6] := 316.3804;
   DATA[1087,8] := 1.0;
   DATA[1087,9] := 1.0;
   DATA[1087,10] := 1.0;
   DATA[1087,11] := 2.010372;
   DATA[1087,13] := 1010.678;
   DATA[1087,14] := 1.0;
   DATA[1087,15] := 1.0;
   DATA[1087,16] := 1.0;
   DATA[1087,17] := 1.0;
   DATA[1087,18] := 1.0;
   DATA[1087,19] := 1.0;
   DATA[1087,20] := 148.808;
   DATA[1087,21] := 154.6526;
   DATA[1087,22] := 1.715952;
   DATA[1087,23] := 881.0433;
   DATA[1087,24] := 2.0;
   DATA[1087,25] := 2.0;
   DATA[1087,26] := 7.879262;
   DATA[1087,27] := 143.5529;
   DATA[1087,28] := 263.0095;
   DATA[1087,29] := 12.07383;
   DATA[1087,30] := 1.724045;
   DATA[1087,31] := 1.300115;
   DATA[1087,32] := 0.7353967;
   DATA[1087,33] := 0.3086827;
   DATA[1087,34] := 2.0;
   DATA[1087,35] := 250.3204;
   DATA[1087,36] := 1.681991;
   DATA[1087,37] := 189.1823;
   DATA[1087,38] := 0.000128152;
   DATA[1087,39] := 1.0;
   DATA[1088,0] := 2.537232;
   DATA[1088,1] := 697.0897;
   DATA[1088,2] := 2.0;
   DATA[1088,3] := 1.0;
   DATA[1088,4] := 262.5288;
   DATA[1088,5] := 8.464369;
   DATA[1088,6] := 316.3804;
   DATA[1088,8] := 1.0;
   DATA[1088,9] := 1.0;
   DATA[1088,10] := 1.0;
   DATA[1088,11] := 2.010372;
   DATA[1088,13] := 1010.758;
   DATA[1088,14] := 1.0;
   DATA[1088,15] := 1.0;
   DATA[1088,16] := 1.0;
   DATA[1088,17] := 1.0;
   DATA[1088,18] := 1.0;
   DATA[1088,19] := 1.0;
   DATA[1088,20] := 148.808;
   DATA[1088,21] := 154.8065;
   DATA[1088,22] := 1.715952;
   DATA[1088,23] := 880.6973;
   DATA[1088,24] := 2.0;
   DATA[1088,25] := 2.0;
   DATA[1088,26] := 7.879262;
   DATA[1088,27] := 143.5529;
   DATA[1088,28] := 263.0095;
   DATA[1088,29] := 12.07383;
   DATA[1088,30] := 1.724045;
   DATA[1088,31] := 1.301396;
   DATA[1088,32] := 0.7353967;
   DATA[1088,33] := 0.3086827;
   DATA[1088,34] := 2.0;
   DATA[1088,35] := 250.3204;
   DATA[1088,36] := 1.585878;
   DATA[1088,37] := 189.0861;
   DATA[1088,38] := 0.000128152;
   DATA[1088,39] := 1.0;
   DATA[1089,0] := 2.537232;
   DATA[1089,1] := 698.0318;
   DATA[1089,2] := 2.0;
   DATA[1089,3] := 1.0;
   DATA[1089,4] := 262.5288;
   DATA[1089,5] := 8.464369;
   DATA[1089,6] := 316.3804;
   DATA[1089,8] := 1.0;
   DATA[1089,9] := 1.0;
   DATA[1089,10] := 1.0;
   DATA[1089,11] := 2.010372;
   DATA[1089,13] := 1010.678;
   DATA[1089,14] := 1.0;
   DATA[1089,15] := 1.0;
   DATA[1089,16] := 1.0;
   DATA[1089,17] := 1.0;
   DATA[1089,18] := 1.0;
   DATA[1089,19] := 1.0;
   DATA[1089,20] := 148.808;
   DATA[1089,21] := 154.8065;
   DATA[1089,22] := 1.715952;
   DATA[1089,23] := 880.6588;
   DATA[1089,24] := 2.0;
   DATA[1089,25] := 2.0;
   DATA[1089,26] := 7.879262;
   DATA[1089,27] := 143.5529;
   DATA[1089,28] := 263.0095;
   DATA[1089,29] := 12.07383;
   DATA[1089,30] := 1.724045;
   DATA[1089,31] := 1.282311;
   DATA[1089,32] := 0.7353967;
   DATA[1089,33] := 0.3086827;
   DATA[1089,34] := 2.0;
   DATA[1089,35] := 250.3204;
   DATA[1089,36] := 1.585878;
   DATA[1089,37] := 189.0861;
   DATA[1089,38] := 0.000128152;
   DATA[1089,39] := 1.0;
   DATA[1090,0] := 2.540435;
   DATA[1090,1] := 698.3851;
   DATA[1090,2] := 2.0;
   DATA[1090,3] := 1.0;
   DATA[1090,4] := 262.5288;
   DATA[1090,5] := 8.464369;
   DATA[1090,6] := 316.3804;
   DATA[1090,8] := 1.0;
   DATA[1090,9] := 1.0;
   DATA[1090,10] := 1.0;
   DATA[1090,11] := 2.010372;
   DATA[1090,13] := 1010.518;
   DATA[1090,14] := 1.0;
   DATA[1090,15] := 1.0;
   DATA[1090,16] := 1.0;
   DATA[1090,17] := 1.0;
   DATA[1090,18] := 1.0;
   DATA[1090,19] := 1.0;
   DATA[1090,20] := 148.808;
   DATA[1090,21] := 154.8065;
   DATA[1090,22] := 1.715952;
   DATA[1090,23] := 879.9282;
   DATA[1090,24] := 2.0;
   DATA[1090,25] := 2.0;
   DATA[1090,26] := 7.879262;
   DATA[1090,27] := 143.5529;
   DATA[1090,28] := 263.0095;
   DATA[1090,29] := 12.07383;
   DATA[1090,30] := 1.724045;
   DATA[1090,31] := 1.276547;
   DATA[1090,32] := 0.7353967;
   DATA[1090,33] := 0.3086827;
   DATA[1090,34] := 2.0;
   DATA[1090,35] := 250.3204;
   DATA[1090,36] := 1.585878;
   DATA[1090,37] := 189.0861;
   DATA[1090,38] := 0.000128152;
   DATA[1090,39] := 1.0;
   DATA[1091,0] := 2.54588;
   DATA[1091,1] := 698.6206;
   DATA[1091,2] := 2.0;
   DATA[1091,3] := 1.0;
   DATA[1091,4] := 262.5288;
   DATA[1091,5] := 8.464369;
   DATA[1091,6] := 316.4829;
   DATA[1091,8] := 1.0;
   DATA[1091,9] := 1.0;
   DATA[1091,10] := 1.0;
   DATA[1091,11] := 2.010372;
   DATA[1091,13] := 1010.919;
   DATA[1091,14] := 1.0;
   DATA[1091,15] := 1.0;
   DATA[1091,16] := 1.0;
   DATA[1091,17] := 1.0;
   DATA[1091,18] := 1.0;
   DATA[1091,19] := 1.0;
   DATA[1091,20] := 148.808;
   DATA[1091,21] := 154.8065;
   DATA[1091,22] := 1.715952;
   DATA[1091,23] := 879.6206;
   DATA[1091,24] := 2.0;
   DATA[1091,25] := 2.0;
   DATA[1091,26] := 7.879262;
   DATA[1091,27] := 143.5529;
   DATA[1091,28] := 263.0095;
   DATA[1091,29] := 12.07383;
   DATA[1091,30] := 1.724045;
   DATA[1091,31] := 1.276547;
   DATA[1091,32] := 0.7353967;
   DATA[1091,33] := 0.3086827;
   DATA[1091,34] := 2.0;
   DATA[1091,35] := 250.3204;
   DATA[1091,36] := 1.585878;
   DATA[1091,37] := 189.0861;
   DATA[1091,38] := 0.000128152;
   DATA[1091,39] := 1.0;
   DATA[1092,0] := 2.551645;
   DATA[1092,1] := 698.8561;
   DATA[1092,2] := 2.0;
   DATA[1092,3] := 1.0;
   DATA[1092,4] := 262.5288;
   DATA[1092,5] := 8.464369;
   DATA[1092,6] := 316.4829;
   DATA[1092,8] := 1.0;
   DATA[1092,9] := 1.0;
   DATA[1092,10] := 1.0;
   DATA[1092,11] := 2.010372;
   DATA[1092,13] := 1010.718;
   DATA[1092,14] := 1.0;
   DATA[1092,15] := 1.0;
   DATA[1092,16] := 1.0;
   DATA[1092,17] := 1.0;
   DATA[1092,18] := 1.0;
   DATA[1092,19] := 1.0;
   DATA[1092,20] := 148.808;
   DATA[1092,21] := 154.8065;
   DATA[1092,22] := 1.715952;
   DATA[1092,23] := 879.2361;
   DATA[1092,24] := 2.0;
   DATA[1092,25] := 2.0;
   DATA[1092,26] := 7.879262;
   DATA[1092,27] := 143.5529;
   DATA[1092,28] := 263.0095;
   DATA[1092,29] := 12.07383;
   DATA[1092,30] := 1.724173;
   DATA[1092,31] := 1.270142;
   DATA[1092,32] := 0.7353967;
   DATA[1092,33] := 0.3086827;
   DATA[1092,34] := 2.0;
   DATA[1092,35] := 250.3204;
   DATA[1092,36] := 1.649953;
   DATA[1092,37] := 189.0861;
   DATA[1092,38] := 0.000128152;
   DATA[1092,39] := 1.0;
   DATA[1093,0] := 2.553566;
   DATA[1093,1] := 699.4841;
   DATA[1093,2] := 2.0;
   DATA[1093,3] := 1.0;
   DATA[1093,4] := 262.5288;
   DATA[1093,5] := 8.464369;
   DATA[1093,6] := 316.4829;
   DATA[1093,8] := 1.0;
   DATA[1093,9] := 1.0;
   DATA[1093,10] := 1.0;
   DATA[1093,11] := 2.010372;
   DATA[1093,13] := 1010.758;
   DATA[1093,14] := 1.0;
   DATA[1093,15] := 1.0;
   DATA[1093,16] := 1.0;
   DATA[1093,17] := 1.0;
   DATA[1093,18] := 1.0;
   DATA[1093,19] := 1.0;
   DATA[1093,20] := 148.808;
   DATA[1093,21] := 154.8065;
   DATA[1093,22] := 1.715952;
   DATA[1093,23] := 879.0054;
   DATA[1093,24] := 2.0;
   DATA[1093,25] := 2.0;
   DATA[1093,26] := 7.877019;
   DATA[1093,27] := 143.5529;
   DATA[1093,28] := 263.0095;
   DATA[1093,29] := 12.07383;
   DATA[1093,30] := 1.72507;
   DATA[1093,31] := 1.270142;
   DATA[1093,32] := 0.7353967;
   DATA[1093,33] := 0.3083624;
   DATA[1093,34] := 2.0;
   DATA[1093,35] := 250.3204;
   DATA[1093,36] := 1.649953;
   DATA[1093,37] := 189.0861;
   DATA[1093,38] := 0.000128152;
   DATA[1093,39] := 1.0;
   DATA[1094,0] := 2.553566;
   DATA[1094,1] := 700.0729;
   DATA[1094,2] := 2.0;
   DATA[1094,3] := 1.0;
   DATA[1094,4] := 262.5288;
   DATA[1094,5] := 8.464369;
   DATA[1094,6] := 316.4829;
   DATA[1094,8] := 1.0;
   DATA[1094,9] := 1.0;
   DATA[1094,10] := 1.0;
   DATA[1094,11] := 2.010372;
   DATA[1094,13] := 1010.758;
   DATA[1094,14] := 1.0;
   DATA[1094,15] := 1.0;
   DATA[1094,16] := 1.0;
   DATA[1094,17] := 1.0;
   DATA[1094,18] := 1.0;
   DATA[1094,19] := 1.0;
   DATA[1094,20] := 148.808;
   DATA[1094,21] := 154.8065;
   DATA[1094,22] := 1.715952;
   DATA[1094,23] := 878.7747;
   DATA[1094,24] := 2.0;
   DATA[1094,25] := 2.0;
   DATA[1094,26] := 7.877019;
   DATA[1094,27] := 143.5529;
   DATA[1094,28] := 263.0095;
   DATA[1094,29] := 12.07383;
   DATA[1094,30] := 1.725968;
   DATA[1094,31] := 1.271295;
   DATA[1094,32] := 0.7353967;
   DATA[1094,33] := 0.3083624;
   DATA[1094,34] := 2.0;
   DATA[1094,35] := 250.3204;
   DATA[1094,36] := 1.649953;
   DATA[1094,37] := 189.0861;
   DATA[1094,38] := 0.000128152;
   DATA[1094,39] := 1.0;
   DATA[1095,0] := 2.547161;
   DATA[1095,1] := 700.6617;
   DATA[1095,2] := 2.0;
   DATA[1095,3] := 1.0;
   DATA[1095,4] := 262.5288;
   DATA[1095,5] := 8.464369;
   DATA[1095,6] := 316.4829;
   DATA[1095,8] := 1.0;
   DATA[1095,9] := 1.0;
   DATA[1095,10] := 1.0;
   DATA[1095,11] := 2.010372;
   DATA[1095,13] := 1010.718;
   DATA[1095,14] := 1.0;
   DATA[1095,15] := 1.0;
   DATA[1095,16] := 1.0;
   DATA[1095,17] := 1.0;
   DATA[1095,18] := 1.0;
   DATA[1095,19] := 1.0;
   DATA[1095,20] := 148.808;
   DATA[1095,21] := 154.8065;
   DATA[1095,22] := 1.715439;
   DATA[1095,23] := 878.2363;
   DATA[1095,24] := 2.0;
   DATA[1095,25] := 2.0;
   DATA[1095,26] := 7.877019;
   DATA[1095,27] := 143.5529;
   DATA[1095,28] := 263.0095;
   DATA[1095,29] := 12.07383;
   DATA[1095,30] := 1.725968;
   DATA[1095,31] := 1.28705;
   DATA[1095,32] := 0.7353967;
   DATA[1095,33] := 0.3083624;
   DATA[1095,34] := 2.0;
   DATA[1095,35] := 250.3204;
   DATA[1095,36] := 1.649953;
   DATA[1095,37] := 189.0861;
   DATA[1095,38] := 0.000128152;
   DATA[1095,39] := 1.0;
   DATA[1096,0] := 2.545559;
   DATA[1096,1] := 701.5253;
   DATA[1096,2] := 2.0;
   DATA[1096,3] := 1.0;
   DATA[1096,4] := 262.5288;
   DATA[1096,5] := 8.464369;
   DATA[1096,6] := 316.4829;
   DATA[1096,8] := 1.0;
   DATA[1096,9] := 1.0;
   DATA[1096,10] := 1.0;
   DATA[1096,11] := 2.010372;
   DATA[1096,13] := 1010.718;
   DATA[1096,14] := 1.0;
   DATA[1096,15] := 1.0;
   DATA[1096,16] := 1.0;
   DATA[1096,17] := 1.0;
   DATA[1096,18] := 1.0;
   DATA[1096,19] := 1.0;
   DATA[1096,20] := 148.808;
   DATA[1096,21] := 154.8065;
   DATA[1096,22] := 1.713389;
   DATA[1096,23] := 877.8134;
   DATA[1096,24] := 2.0;
   DATA[1096,25] := 2.0;
   DATA[1096,26] := 7.877019;
   DATA[1096,27] := 143.5529;
   DATA[1096,28] := 263.0095;
   DATA[1096,29] := 12.07383;
   DATA[1096,30] := 1.725968;
   DATA[1096,31] := 1.284873;
   DATA[1096,32] := 0.7353967;
   DATA[1096,33] := 0.306761;
   DATA[1096,34] := 2.0;
   DATA[1096,35] := 250.3204;
   DATA[1096,36] := 1.649953;
   DATA[1096,37] := 189.0861;
   DATA[1096,38] := 0.000128152;
   DATA[1096,39] := 1.0;
   DATA[1097,0] := 2.545559;
   DATA[1097,1] := 702.1926;
   DATA[1097,2] := 2.0;
   DATA[1097,3] := 1.0;
   DATA[1097,4] := 262.5288;
   DATA[1097,5] := 8.464369;
   DATA[1097,6] := 316.4829;
   DATA[1097,8] := 1.0;
   DATA[1097,9] := 1.0;
   DATA[1097,10] := 1.0;
   DATA[1097,11] := 2.010372;
   DATA[1097,13] := 1010.718;
   DATA[1097,14] := 1.0;
   DATA[1097,15] := 1.0;
   DATA[1097,16] := 1.0;
   DATA[1097,17] := 1.0;
   DATA[1097,18] := 1.0;
   DATA[1097,19] := 1.0;
   DATA[1097,20] := 148.808;
   DATA[1097,21] := 154.7808;
   DATA[1097,22] := 1.713389;
   DATA[1097,23] := 876.8906;
   DATA[1097,24] := 2.0;
   DATA[1097,25] := 2.0;
   DATA[1097,26] := 7.877019;
   DATA[1097,27] := 143.5529;
   DATA[1097,28] := 263.0095;
   DATA[1097,29] := 12.07383;
   DATA[1097,30] := 1.725968;
   DATA[1097,31] := 1.286922;
   DATA[1097,32] := 0.7353967;
   DATA[1097,33] := 0.306761;
   DATA[1097,34] := 2.0;
   DATA[1097,35] := 250.3204;
   DATA[1097,36] := 1.649953;
   DATA[1097,37] := 189.2143;
   DATA[1097,38] := 0.000128152;
   DATA[1097,39] := 1.0;
   DATA[1098,0] := 2.543317;
   DATA[1098,1] := 702.9777;
   DATA[1098,2] := 2.0;
   DATA[1098,3] := 1.0;
   DATA[1098,4] := 262.5288;
   DATA[1098,5] := 8.463408;
   DATA[1098,6] := 316.4829;
   DATA[1098,8] := 1.0;
   DATA[1098,9] := 1.0;
   DATA[1098,10] := 1.0;
   DATA[1098,11] := 2.010372;
   DATA[1098,13] := 1010.959;
   DATA[1098,14] := 1.0;
   DATA[1098,15] := 1.0;
   DATA[1098,16] := 1.0;
   DATA[1098,17] := 1.0;
   DATA[1098,18] := 1.0;
   DATA[1098,19] := 1.0;
   DATA[1098,20] := 148.808;
   DATA[1098,21] := 154.6783;
   DATA[1098,22] := 1.713389;
   DATA[1098,23] := 876.5445;
   DATA[1098,24] := 2.0;
   DATA[1098,25] := 2.0;
   DATA[1098,26] := 7.878942;
   DATA[1098,27] := 143.5529;
   DATA[1098,28] := 263.0095;
   DATA[1098,29] := 12.07383;
   DATA[1098,30] := 1.725968;
   DATA[1098,31] := 1.285769;
   DATA[1098,32] := 0.7353967;
   DATA[1098,33] := 0.3083624;
   DATA[1098,34] := 2.0;
   DATA[1098,35] := 250.3204;
   DATA[1098,36] := 1.649953;
   DATA[1098,37] := 189.2143;
   DATA[1098,38] := 0.000128152;
   DATA[1098,39] := 1.0;
   DATA[1099,0] := 2.543317;
   DATA[1099,1] := 703.5272;
   DATA[1099,2] := 2.0;
   DATA[1099,3] := 1.0;
   DATA[1099,4] := 262.5288;
   DATA[1099,5] := 8.461164;
   DATA[1099,6] := 316.4829;
   DATA[1099,8] := 1.0;
   DATA[1099,9] := 1.0;
   DATA[1099,10] := 1.0;
   DATA[1099,11] := 2.010372;
   DATA[1099,13] := 1011.239;
   DATA[1099,14] := 1.0;
   DATA[1099,15] := 1.0;
   DATA[1099,16] := 1.0;
   DATA[1099,17] := 1.0;
   DATA[1099,18] := 1.0;
   DATA[1099,19] := 1.0;
   DATA[1099,20] := 148.808;
   DATA[1099,21] := 154.6783;
   DATA[1099,22] := 1.713389;
   DATA[1099,23] := 876.2369;
   DATA[1099,24] := 2.0;
   DATA[1099,25] := 2.0;
   DATA[1099,26] := 7.879262;
   DATA[1099,27] := 143.5529;
   DATA[1099,28] := 263.0095;
   DATA[1099,29] := 12.07383;
   DATA[1099,30] := 1.725968;
   DATA[1099,31] := 1.28167;
   DATA[1099,32] := 0.7353967;
   DATA[1099,33] := 0.3083624;
   DATA[1099,34] := 2.0;
   DATA[1099,35] := 250.3204;
   DATA[1099,36] := 1.649953;
   DATA[1099,37] := 189.2143;
   DATA[1099,38] := 0.000128152;
   DATA[1099,39] := 1.0;
   DATA[1100,0] := 2.543317;
   DATA[1100,1] := 704.1945;
   DATA[1100,2] := 2.0;
   DATA[1100,3] := 1.0;
   DATA[1100,4] := 262.5288;
   DATA[1100,5] := 8.461164;
   DATA[1100,6] := 316.4829;
   DATA[1100,8] := 1.0;
   DATA[1100,9] := 1.0;
   DATA[1100,10] := 1.0;
   DATA[1100,11] := 2.010372;
   DATA[1100,13] := 1010.839;
   DATA[1100,14] := 1.0;
   DATA[1100,15] := 1.0;
   DATA[1100,16] := 1.0;
   DATA[1100,17] := 1.0;
   DATA[1100,18] := 1.0;
   DATA[1100,19] := 1.0;
   DATA[1100,20] := 148.808;
   DATA[1100,21] := 154.5757;
   DATA[1100,22] := 1.714158;
   DATA[1100,23] := 875.9293;
   DATA[1100,24] := 2.0;
   DATA[1100,25] := 2.0;
   DATA[1100,26] := 7.879262;
   DATA[1100,27] := 143.5529;
   DATA[1100,28] := 263.0095;
   DATA[1100,29] := 12.07383;
   DATA[1100,30] := 1.724173;
   DATA[1100,31] := 1.28167;
   DATA[1100,32] := 0.7353967;
   DATA[1100,33] := 0.3074656;
   DATA[1100,34] := 2.0;
   DATA[1100,35] := 250.3204;
   DATA[1100,36] := 1.649953;
   DATA[1100,37] := 188.974;
   DATA[1100,38] := 0.000128152;
   DATA[1100,39] := 1.0;
   DATA[1101,0] := 2.543317;
   DATA[1101,1] := 704.7833;
   DATA[1101,2] := 2.0;
   DATA[1101,3] := 1.0;
   DATA[1101,4] := 262.5288;
   DATA[1101,5] := 8.461164;
   DATA[1101,6] := 316.4829;
   DATA[1101,8] := 1.0;
   DATA[1101,9] := 1.0;
   DATA[1101,10] := 1.0;
   DATA[1101,11] := 2.010372;
   DATA[1101,13] := 1010.718;
   DATA[1101,14] := 1.0;
   DATA[1101,15] := 1.0;
   DATA[1101,16] := 1.0;
   DATA[1101,17] := 1.0;
   DATA[1101,18] := 1.0;
   DATA[1101,19] := 1.0;
   DATA[1101,20] := 148.808;
   DATA[1101,21] := 154.5757;
   DATA[1101,22] := 1.715311;
   DATA[1101,23] := 875.9677;
   DATA[1101,24] := 2.0;
   DATA[1101,25] := 2.0;
   DATA[1101,26] := 7.879262;
   DATA[1101,27] := 143.5529;
   DATA[1101,28] := 263.0095;
   DATA[1101,29] := 12.07383;
   DATA[1101,30] := 1.724173;
   DATA[1101,31] := 1.271551;
   DATA[1101,32] := 0.7353967;
   DATA[1101,33] := 0.3077859;
   DATA[1101,34] := 2.0;
   DATA[1101,35] := 250.1923;
   DATA[1101,36] := 1.649953;
   DATA[1101,37] := 188.974;
   DATA[1101,38] := 0.000128152;
   DATA[1101,39] := 1.0;
   DATA[1102,0] := 2.553566;
   DATA[1102,1] := 705.5291;
   DATA[1102,2] := 2.0;
   DATA[1102,3] := 1.0;
   DATA[1102,4] := 262.5288;
   DATA[1102,5] := 8.462126;
   DATA[1102,6] := 316.4829;
   DATA[1102,8] := 1.0;
   DATA[1102,9] := 1.0;
   DATA[1102,10] := 1.0;
   DATA[1102,11] := 2.010372;
   DATA[1102,13] := 1010.718;
   DATA[1102,14] := 1.0;
   DATA[1102,15] := 1.0;
   DATA[1102,16] := 1.0;
   DATA[1102,17] := 1.0;
   DATA[1102,18] := 1.0;
   DATA[1102,19] := 1.0;
   DATA[1102,20] := 148.808;
   DATA[1102,21] := 154.5757;
   DATA[1102,22] := 1.715439;
   DATA[1102,23] := 875.4678;
   DATA[1102,24] := 2.0;
   DATA[1102,25] := 2.0;
   DATA[1102,26] := 7.879262;
   DATA[1102,27] := 143.5529;
   DATA[1102,28] := 263.0095;
   DATA[1102,29] := 12.07383;
   DATA[1102,30] := 1.724173;
   DATA[1102,31] := 1.276162;
   DATA[1102,32] := 0.7353967;
   DATA[1102,33] := 0.3084265;
   DATA[1102,34] := 2.0;
   DATA[1102,35] := 250.1762;
   DATA[1102,36] := 1.649953;
   DATA[1102,37] := 188.974;
   DATA[1102,38] := 0.000128152;
   DATA[1102,39] := 1.0;
   DATA[1103,0] := 2.553566;
   DATA[1103,1] := 706.2356;
   DATA[1103,2] := 2.0;
   DATA[1103,3] := 1.0;
   DATA[1103,4] := 262.5288;
   DATA[1103,5] := 8.463728;
   DATA[1103,6] := 316.4829;
   DATA[1103,8] := 1.0;
   DATA[1103,9] := 1.0;
   DATA[1103,10] := 1.0;
   DATA[1103,11] := 2.010372;
   DATA[1103,13] := 1010.879;
   DATA[1103,14] := 1.0;
   DATA[1103,15] := 1.0;
   DATA[1103,16] := 1.0;
   DATA[1103,17] := 1.0;
   DATA[1103,18] := 1.0;
   DATA[1103,19] := 1.0;
   DATA[1103,20] := 148.808;
   DATA[1103,21] := 154.5757;
   DATA[1103,22] := 1.715439;
   DATA[1103,23] := 875.2756;
   DATA[1103,24] := 2.0;
   DATA[1103,25] := 2.0;
   DATA[1103,26] := 7.879262;
   DATA[1103,27] := 143.5529;
   DATA[1103,28] := 263.0095;
   DATA[1103,29] := 12.07383;
   DATA[1103,30] := 1.725327;
   DATA[1103,31] := 1.276162;
   DATA[1103,32] := 0.7353967;
   DATA[1103,33] := 0.3086827;
   DATA[1103,34] := 2.0;
   DATA[1103,35] := 250.1762;
   DATA[1103,36] := 1.649953;
   DATA[1103,37] := 188.974;
   DATA[1103,38] := 0.000128152;
   DATA[1103,39] := 1.0;
   DATA[1104,0] := 2.553566;
   DATA[1104,1] := 706.5496;
   DATA[1104,2] := 2.0;
   DATA[1104,3] := 1.0;
   DATA[1104,4] := 262.5288;
   DATA[1104,5] := 8.464369;
   DATA[1104,6] := 316.4829;
   DATA[1104,8] := 1.0;
   DATA[1104,9] := 1.0;
   DATA[1104,10] := 1.0;
   DATA[1104,11] := 2.010372;
   DATA[1104,13] := 1010.638;
   DATA[1104,14] := 1.0;
   DATA[1104,15] := 1.0;
   DATA[1104,16] := 1.0;
   DATA[1104,17] := 1.0;
   DATA[1104,18] := 1.0;
   DATA[1104,19] := 1.0;
   DATA[1104,20] := 148.808;
   DATA[1104,21] := 154.5757;
   DATA[1104,22] := 1.715824;
   DATA[1104,23] := 874.8141;
   DATA[1104,24] := 2.0;
   DATA[1104,25] := 2.0;
   DATA[1104,26] := 7.879262;
   DATA[1104,27] := 143.5529;
   DATA[1104,28] := 263.0095;
   DATA[1104,29] := 12.07383;
   DATA[1104,30] := 1.725327;
   DATA[1104,31] := 1.275778;
   DATA[1104,32] := 0.7353967;
   DATA[1104,33] := 0.3086827;
   DATA[1104,34] := 2.0;
   DATA[1104,35] := 250.1762;
   DATA[1104,36] := 1.649953;
   DATA[1104,37] := 188.974;
   DATA[1104,38] := 0.000128152;
   DATA[1104,39] := 1.0;
   DATA[1105,0] := 2.554847;
   DATA[1105,1] := 707.4917;
   DATA[1105,2] := 2.0;
   DATA[1105,3] := 1.0;
   DATA[1105,4] := 262.5288;
   DATA[1105,5] := 8.464369;
   DATA[1105,6] := 316.4829;
   DATA[1105,8] := 1.0;
   DATA[1105,9] := 1.0;
   DATA[1105,10] := 1.0;
   DATA[1105,11] := 2.010372;
   DATA[1105,13] := 1011.119;
   DATA[1105,14] := 1.0;
   DATA[1105,15] := 1.0;
   DATA[1105,16] := 1.0;
   DATA[1105,17] := 1.0;
   DATA[1105,18] := 1.0;
   DATA[1105,19] := 1.0;
   DATA[1105,20] := 148.808;
   DATA[1105,21] := 154.5757;
   DATA[1105,22] := 1.715824;
   DATA[1105,23] := 874.5834;
   DATA[1105,24] := 2.0;
   DATA[1105,25] := 2.0;
   DATA[1105,26] := 7.879262;
   DATA[1105,27] := 143.5529;
   DATA[1105,28] := 263.0095;
   DATA[1105,29] := 12.07383;
   DATA[1105,30] := 1.725327;
   DATA[1105,31] := 1.290765;
   DATA[1105,32] := 0.7353967;
   DATA[1105,33] := 0.3086827;
   DATA[1105,34] := 2.0;
   DATA[1105,35] := 250.1762;
   DATA[1105,36] := 1.649953;
   DATA[1105,37] := 188.974;
   DATA[1105,38] := 0.000128152;
   DATA[1105,39] := 1.0;
   DATA[1106,0] := 2.554847;
   DATA[1106,1] := 708.1982;
   DATA[1106,2] := 2.0;
   DATA[1106,3] := 1.0;
   DATA[1106,4] := 262.5288;
   DATA[1106,5] := 8.464369;
   DATA[1106,6] := 316.4829;
   DATA[1106,8] := 1.0;
   DATA[1106,9] := 1.0;
   DATA[1106,10] := 1.0;
   DATA[1106,11] := 2.010372;
   DATA[1106,13] := 1011.119;
   DATA[1106,14] := 1.0;
   DATA[1106,15] := 1.0;
   DATA[1106,16] := 1.0;
   DATA[1106,17] := 1.0;
   DATA[1106,18] := 1.0;
   DATA[1106,19] := 1.0;
   DATA[1106,20] := 148.808;
   DATA[1106,21] := 154.5757;
   DATA[1106,22] := 1.717489;
   DATA[1106,23] := 874.122;
   DATA[1106,24] := 2.0;
   DATA[1106,25] := 2.0;
   DATA[1106,26] := 7.879262;
   DATA[1106,27] := 143.5529;
   DATA[1106,28] := 263.0095;
   DATA[1106,29] := 12.07383;
   DATA[1106,30] := 1.724173;
   DATA[1106,31] := 1.289612;
   DATA[1106,32] := 0.7353967;
   DATA[1106,33] := 0.3086827;
   DATA[1106,34] := 2.0;
   DATA[1106,35] := 250.1762;
   DATA[1106,36] := 1.762086;
   DATA[1106,37] := 189.0861;
   DATA[1106,38] := 0.000128152;
   DATA[1106,39] := 1.0;
   DATA[1107,0] := 2.554847;
   DATA[1107,1] := 708.4338;
   DATA[1107,2] := 2.0;
   DATA[1107,3] := 1.0;
   DATA[1107,4] := 262.5288;
   DATA[1107,5] := 8.464369;
   DATA[1107,6] := 316.5342;
   DATA[1107,8] := 1.0;
   DATA[1107,9] := 1.0;
   DATA[1107,10] := 1.0;
   DATA[1107,11] := 2.010372;
   DATA[1107,13] := 1011.079;
   DATA[1107,14] := 1.0;
   DATA[1107,15] := 1.0;
   DATA[1107,16] := 1.0;
   DATA[1107,17] := 1.0;
   DATA[1107,18] := 1.0;
   DATA[1107,19] := 1.0;
   DATA[1107,20] := 148.808;
   DATA[1107,21] := 154.5757;
   DATA[1107,22] := 1.717489;
   DATA[1107,23] := 874.122;
   DATA[1107,24] := 2.0;
   DATA[1107,25] := 2.0;
   DATA[1107,26] := 7.879262;
   DATA[1107,27] := 143.6042;
   DATA[1107,28] := 263.0095;
   DATA[1107,29] := 12.07383;
   DATA[1107,30] := 1.723789;
   DATA[1107,31] := 1.286282;
   DATA[1107,32] := 0.7374452;
   DATA[1107,33] := 0.3086827;
   DATA[1107,34] := 2.0;
   DATA[1107,35] := 250.1762;
   DATA[1107,36] := 1.762086;
   DATA[1107,37] := 189.0861;
   DATA[1107,38] := 0.000128152;
   DATA[1107,39] := 1.0;
   DATA[1108,0] := 2.545559;
   DATA[1108,1] := 709.2974;
   DATA[1108,2] := 2.0;
   DATA[1108,3] := 1.0;
   DATA[1108,4] := 262.5288;
   DATA[1108,5] := 8.464369;
   DATA[1108,6] := 316.5342;
   DATA[1108,8] := 1.0;
   DATA[1108,9] := 1.0;
   DATA[1108,10] := 1.0;
   DATA[1108,11] := 2.010372;
   DATA[1108,12] := 0.000256221;
   DATA[1108,13] := 1011.279;
   DATA[1108,14] := 1.0;
   DATA[1108,15] := 1.0;
   DATA[1108,16] := 1.0;
   DATA[1108,17] := 1.0;
   DATA[1108,18] := 1.0;
   DATA[1108,19] := 1.0;
   DATA[1108,20] := 148.808;
   DATA[1108,21] := 154.5757;
   DATA[1108,22] := 1.71608;
   DATA[1108,23] := 874.0451;
   DATA[1108,24] := 2.0;
   DATA[1108,25] := 2.0;
   DATA[1108,26] := 7.879262;
   DATA[1108,27] := 143.6042;
   DATA[1108,28] := 263.0095;
   DATA[1108,29] := 12.07383;
   DATA[1108,30] := 1.723789;
   DATA[1108,31] := 1.286666;
   DATA[1108,32] := 0.7383414;
   DATA[1108,33] := 0.3086827;
   DATA[1108,34] := 2.0;
   DATA[1108,35] := 250.1762;
   DATA[1108,36] := 1.762086;
   DATA[1108,37] := 189.0861;
   DATA[1108,38] := 0.000128152;
   DATA[1108,39] := 1.0;
   DATA[1109,0] := 2.543317;
   DATA[1109,1] := 709.6114;
   DATA[1109,2] := 2.0;
   DATA[1109,3] := 1.0;
   DATA[1109,4] := 262.5288;
   DATA[1109,5] := 8.464369;
   DATA[1109,6] := 316.5342;
   DATA[1109,8] := 1.0;
   DATA[1109,9] := 1.0;
   DATA[1109,10] := 1.0;
   DATA[1109,11] := 2.010372;
   DATA[1109,12] := 0.000256221;
   DATA[1109,13] := 1010.758;
   DATA[1109,14] := 1.0;
   DATA[1109,15] := 1.0;
   DATA[1109,16] := 1.0;
   DATA[1109,17] := 1.0;
   DATA[1109,18] := 1.0;
   DATA[1109,19] := 1.0;
   DATA[1109,20] := 148.808;
   DATA[1109,21] := 154.5757;
   DATA[1109,22] := 1.71608;
   DATA[1109,23] := 873.4683;
   DATA[1109,24] := 2.0;
   DATA[1109,25] := 2.0;
   DATA[1109,26] := 7.879262;
   DATA[1109,27] := 143.6042;
   DATA[1109,28] := 263.0095;
   DATA[1109,29] := 12.07383;
   DATA[1109,30] := 1.723789;
   DATA[1109,31] := 1.272832;
   DATA[1109,32] := 0.7383414;
   DATA[1109,33] := 0.3086827;
   DATA[1109,34] := 2.0;
   DATA[1109,35] := 250.3525;
   DATA[1109,36] := 1.762086;
   DATA[1109,37] := 189.0861;
   DATA[1109,38] := 0.000128152;
   DATA[1109,39] := 1.0;
   DATA[1110,0] := 2.540435;
   DATA[1110,1] := 710.2394;
   DATA[1110,2] := 2.0;
   DATA[1110,3] := 1.0;
   DATA[1110,4] := 262.5288;
   DATA[1110,5] := 8.464369;
   DATA[1110,6] := 316.5342;
   DATA[1110,8] := 1.0;
   DATA[1110,9] := 1.0;
   DATA[1110,10] := 1.0;
   DATA[1110,11] := 2.010372;
   DATA[1110,12] := 0.000256221;
   DATA[1110,13] := 1011.079;
   DATA[1110,14] := 1.0;
   DATA[1110,15] := 1.0;
   DATA[1110,16] := 1.0;
   DATA[1110,17] := 1.0;
   DATA[1110,18] := 1.0;
   DATA[1110,19] := 1.0;
   DATA[1110,20] := 148.808;
   DATA[1110,21] := 154.5757;
   DATA[1110,22] := 1.71608;
   DATA[1110,23] := 873.2376;
   DATA[1110,24] := 2.0;
   DATA[1110,25] := 2.0;
   DATA[1110,26] := 7.879262;
   DATA[1110,27] := 143.6042;
   DATA[1110,28] := 263.0095;
   DATA[1110,29] := 12.07383;
   DATA[1110,30] := 1.723789;
   DATA[1110,31] := 1.276803;
   DATA[1110,32] := 0.7383414;
   DATA[1110,33] := 0.3084265;
   DATA[1110,34] := 2.0;
   DATA[1110,35] := 250.3525;
   DATA[1110,36] := 1.762086;
   DATA[1110,37] := 189.0861;
   DATA[1110,38] := 0.000128152;
   DATA[1110,39] := 1.0;
   DATA[1111,0] := 2.540435;
   DATA[1111,1] := 711.1422;
   DATA[1111,2] := 2.0;
   DATA[1111,3] := 1.0;
   DATA[1111,4] := 262.5288;
   DATA[1111,5] := 8.464048;
   DATA[1111,6] := 316.5342;
   DATA[1111,8] := 1.0;
   DATA[1111,9] := 1.0;
   DATA[1111,10] := 1.0;
   DATA[1111,11] := 2.010372;
   DATA[1111,12] := 0.000256221;
   DATA[1111,13] := 1010.919;
   DATA[1111,14] := 1.0;
   DATA[1111,15] := 1.0;
   DATA[1111,16] := 1.0;
   DATA[1111,17] := 1.0;
   DATA[1111,18] := 1.0;
   DATA[1111,19] := 1.0;
   DATA[1111,20] := 148.808;
   DATA[1111,21] := 154.5757;
   DATA[1111,22] := 1.71608;
   DATA[1111,23] := 873.353;
   DATA[1111,24] := 2.0;
   DATA[1111,25] := 2.0;
   DATA[1111,26] := 7.879262;
   DATA[1111,27] := 143.6042;
   DATA[1111,28] := 263.0095;
   DATA[1111,29] := 12.07383;
   DATA[1111,30] := 1.726865;
   DATA[1111,31] := 1.270014;
   DATA[1111,32] := 0.7383414;
   DATA[1111,33] := 0.3084265;
   DATA[1111,34] := 2.0;
   DATA[1111,35] := 250.3525;
   DATA[1111,36] := 1.762086;
   DATA[1111,37] := 189.0861;
   DATA[1111,38] := 0.000128152;
   DATA[1111,39] := 1.0;
   DATA[1112,0] := 2.540435;
   DATA[1112,1] := 711.2207;
   DATA[1112,2] := 2.0;
   DATA[1112,3] := 1.0;
   DATA[1112,4] := 262.5288;
   DATA[1112,5] := 8.462446;
   DATA[1112,6] := 316.5342;
   DATA[1112,8] := 1.0;
   DATA[1112,9] := 1.0;
   DATA[1112,10] := 1.0;
   DATA[1112,11] := 2.010372;
   DATA[1112,12] := 0.000256221;
   DATA[1112,13] := 1011.239;
   DATA[1112,14] := 1.0;
   DATA[1112,15] := 1.0;
   DATA[1112,16] := 1.0;
   DATA[1112,17] := 1.0;
   DATA[1112,18] := 1.0;
   DATA[1112,19] := 1.0;
   DATA[1112,20] := 148.808;
   DATA[1112,21] := 154.5757;
   DATA[1112,22] := 1.71608;
   DATA[1112,23] := 872.6993;
   DATA[1112,24] := 2.0;
   DATA[1112,25] := 2.0;
   DATA[1112,26] := 7.879262;
   DATA[1112,27] := 143.6042;
   DATA[1112,28] := 263.0095;
